(* Logix 5000 project; controller Sucrose_Main Emulate 5570 rev 20.12; software revision 20.01; part 2 of 30 *)

ADD_ON_INSTRUCTION QSI_Discrete_Device   (* revision 2.0 *)
// Revision note:
// Combined Discrete and Motor Starters into Single AOI
// Combined Feedback and No Feedback into Single AOI
// Added Config Param to select Feedback/No Feedback
// Added Config Param to Disable Output During Alarm
// Added Config Param to select "Energize"/"Start" Text
// Added Manual On Reset Logic During Alarm
// Added Zone & Device Specific Alarm Ack Logic
// Added Zone Manual Mode Enable Logic
// Help:
// Discrete Outputs Devices such as:
// Motors and Pumps on Starters, Solenoid Valves (Non FV and Non Analog Controlled), Beacons, Horns, Solenoids, etc.
VAR_OUTPUT
   DO_Energize : BOOL; {required}   // Alias to OutputCard to Energize DO
END_VAR
VAR_INPUT
   DI_Energized_Feedback : BOOL; {required}   // Alias to Input Card to Confirm Device is Energized
   DI_Disconnect_OK_Feedback : BOOL; {required}   // Alias to Input Card to Confirm Disconnect is OK
   ALM_ACK : BOOL; {required}   // Alias to Zone Master Alarm Acknowledge
   MM_Enable : BOOL; {required}   // Alias to Zone Master Manual Mode Enable
   Config_Energized_Feedback : BOOL := 1; {visible}   // Config Whether Device has Energized Feedback (0= No, 1= Yes) Note: Alarm Disabled if No Feedback
   Config_Disconnect_Feedback : BOOL := 1; {visible}   // Config Whether Device has Disconnect Feedback (0 = No, 1 = Yes)
   Config_Energized_Text : BOOL := 1; {visible}   // Configure Device HMI Popup Text (0="Started" {Motors, Pumps}; 1="Energized" {Most Devices}
   Config_MO_ResetOnAlarm : BOOL := 1; {visible}   // Configure Whether .MO Bit Turns Off when Device Alarm Condition Exists
   Config_OutputDisable_OnAlarm : BOOL; {visible}   // Configure Whether Device OutputTurns Off when Device Alarm Condition Exists
   Config_TMR_Alm_Preset_ms : DINT; {visible}   // Configure Device AlarmTimer Preset In Milliseconds
   Config_TMR_Off_Preset_ms : DINT; {visible}   // Configure Delay Stop Timer Preset In Milliseconds
   Config_TMR_On_Preset_ms : DINT; {visible}   // Configure Delay Start Timer Preset In Milliseconds
   HMI_MM : BOOL; {visible}   // Manual Mode Bit From HMI
   HMI_MO : BOOL; {visible}   // Manual On Bit From HMI
   HMI_ALM_ACK : BOOL;   // AOI Device Specific Alarm Acknowledge From HMI
END_VAR
VAR_OUTPUT
   HMI_Alarmed : BOOL;   // Alarm Status To HMI
   HMI_Energized : BOOL;   // Energized Status To HMI
   HMI_Disconnect_OK : BOOL;   // Disconnect Off Status To HMI
END_VAR
VAR_INPUT
   Energize_Permissive : BOOL;   // Energize Permissive Interlock From Logic
   Energize_Enable : BOOL;   // Energize Enable Interlock From Logic
END_VAR
VAR_OUTPUT
   ALM : BOOL; {visible}   // Device Alarm
END_VAR
VAR_INPUT
   Comment : BOOL;   // Comment for Description Rung to Start Each Routine
   Unused_Input_BOOL : BOOL;   // Trash Tag For Required AOI Input Variables That Are Unused for Current Device (Type Boolean)
END_VAR
VAR_OUTPUT
   Unused_Output_BOOL : BOOL;   // Trash Tag For Required AOI Output Variables That Are Unused for Current Device (Type Boolean)
END_VAR
VAR
   ONS : BOOL[32];
   TMR_Alm : TIMER; {access None}
   TMR_On : TIMER; {access None}
   TMR_Off : TIMER; {access None}
END_VAR

ROUTINE Logic   (* ladder *)
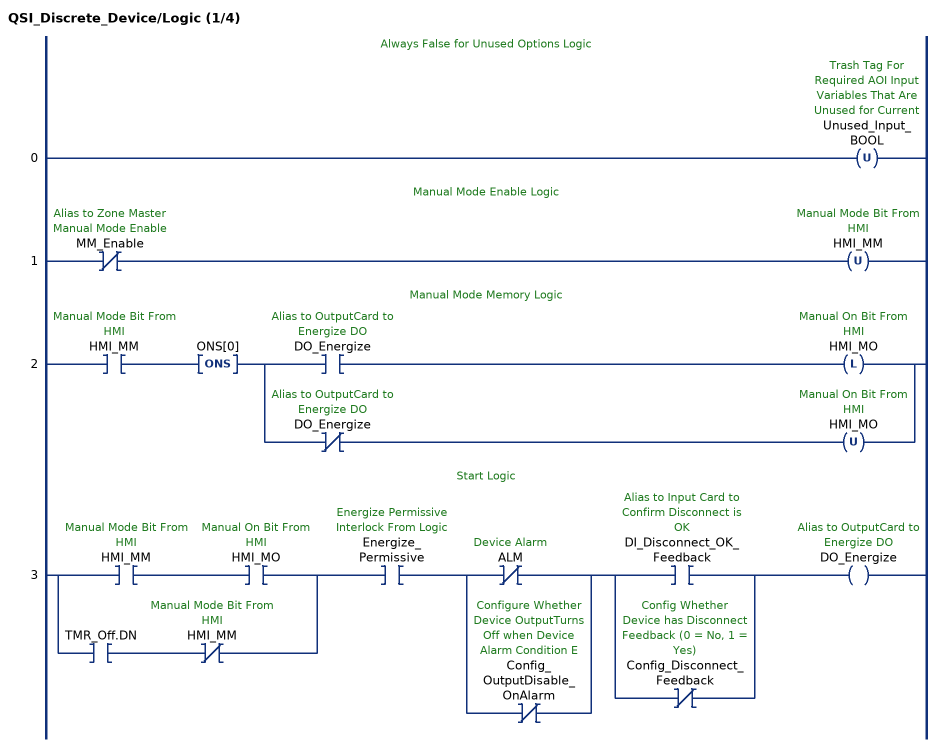
   // Always False for Unused Options Logic
   0: OTU(Unused_Input_BOOL);
   // Manual Mode Enable Logic
   1: XIO(MM_Enable)OTU(HMI_MM);
   // Manual Mode Memory Logic
   2: XIC(HMI_MM)ONS(ONS[0])[XIC(DO_Energize) OTL(HMI_MO) ,XIO(DO_Energize) OTU(HMI_MO) ];
   // Start Logic
   3: [XIC(HMI_MM) XIC(HMI_MO) ,XIC(TMR_Off.DN) XIO(HMI_MM) ]XIC(Energize_Permissive)[XIO(ALM) ,XIO(Config_OutputDisable_OnAlarm) ][XIC(DI_Disconnect_OK_Feedback) ,XIO(Config_Disconnect_Feedback) ]OTE(DO_Energize);
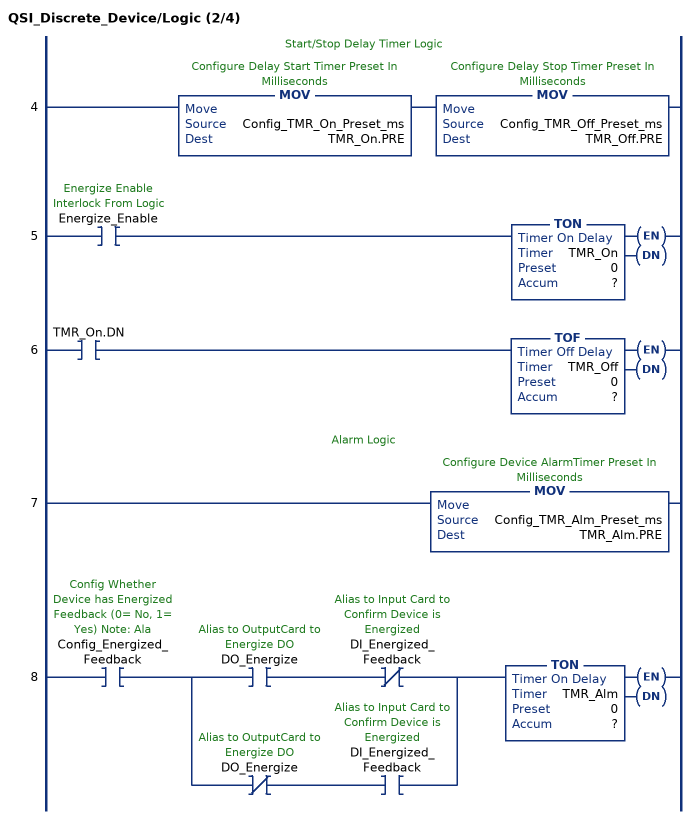
   // Start/Stop Delay Timer Logic
   4: MOV(Config_TMR_On_Preset_ms,TMR_On.PRE)MOV(Config_TMR_Off_Preset_ms,TMR_Off.PRE);
   5: XIC(Energize_Enable)TON(TMR_On,?,?);
   6: XIC(TMR_On.DN)TOF(TMR_Off,?,?);
   // Alarm Logic
   7: MOV(Config_TMR_Alm_Preset_ms,TMR_Alm.PRE);
   8: XIC(Config_Energized_Feedback)[XIC(DO_Energize) XIO(DI_Energized_Feedback) ,XIO(DO_Energize) XIC(DI_Energized_Feedback) ]TON(TMR_Alm,?,?);
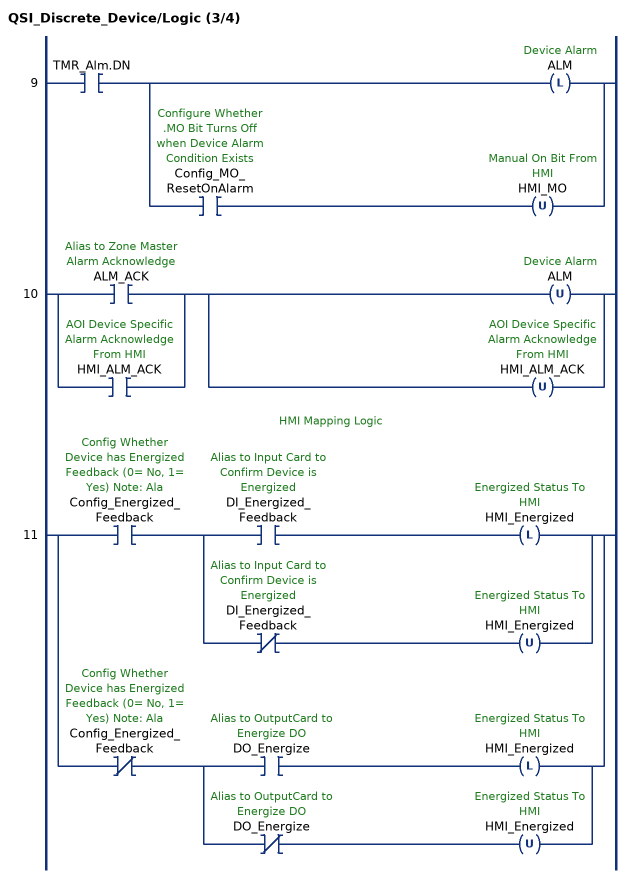
   9: XIC(TMR_Alm.DN)[OTL(ALM) ,XIC(Config_MO_ResetOnAlarm) OTU(HMI_MO) ];
   10: [XIC(ALM_ACK) ,XIC(HMI_ALM_ACK) ][OTU(ALM) ,OTU(HMI_ALM_ACK) ];
   // HMI Mapping Logic
   11: [XIC(Config_Energized_Feedback) [XIC(DI_Energized_Feedback) OTL(HMI_Energized) ,XIO(DI_Energized_Feedback) OTU(HMI_Energized) ] ,XIO(Config_Energized_Feedback) [XIC(DO_Energize) OTL(HMI_Energized) ,XIO(DO_Energize) OTU(HMI_Energized) ] ];
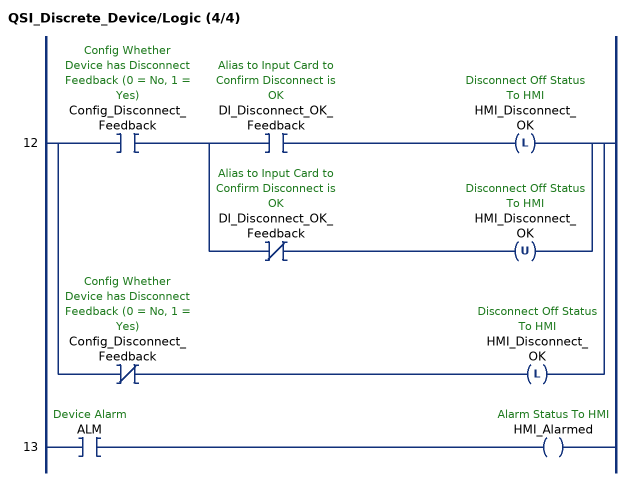
   12: [XIC(Config_Disconnect_Feedback) [XIC(DI_Disconnect_OK_Feedback) OTL(HMI_Disconnect_OK) ,XIO(DI_Disconnect_OK_Feedback) OTU(HMI_Disconnect_OK) ] ,XIO(Config_Disconnect_Feedback) OTL(HMI_Disconnect_OK) ];
   13: XIC(ALM)OTE(HMI_Alarmed);
END_ROUTINE
END_ADD_ON_INSTRUCTION

ADD_ON_INSTRUCTION QSI_Flow_Valve   (* revision 2.0 *)
// Revision note:
// Combined al Non-Analog Flow Valves  into Single AOI
// Combined Feedback and No Feedback into Single AOI
// Added Config Param to select N.O. or N.C. Valve
// Added Config Param to select Opened & Closed Feedback or No Feedback
// Added Manual On Reset Logic During Alarm
// Added Zone & Device Specific Alarm Ack Logic
// Added Zone Manual Mode Enable Logic
// Help:
// Discrete Flow Valves with and without feedback, and with and without Seat Lifts such as:
// Mix Proof, Stop Valves, and other Flow Valves
VAR_OUTPUT
   DO_Energize : BOOL; {required}   // Alias to OutputCard to Energize DO
   DO_USL_Energize : BOOL; {required}   // Alias to OutputCard to Energize Upper Seat Lift DO
   DO_LSL_Energize : BOOL; {required}   // Alias to OutputCard to Energize Lower Seat Lift DO
END_VAR
VAR_INPUT
   DI_Opened_Feedback : BOOL; {required}   // Alias to Input Card to Confirm Device is at Opened Position
   DI_Closed_Feedback : BOOL; {required}   // Alias to Input Card to Confirm Device is at Closed Position
   ALM_ACK : BOOL; {required}   // Alias to Zone Master Alarm Acknowledge
   MM_Enable : BOOL; {required}   // Alias to Zone Master Manual Mode Enable
   Config_NO_Valve : BOOL; {visible}   // Configure Whether Valve is Normally Closed (0 = N.C., 1 = N.O.)
   Config_Opened_Feedback : BOOL := 1; {visible}   // Config Whether Device has Opened Feedback (0= No, 1= Yes) Note: Alarm Disabled if No Feedback
   Config_Closed_Feedback : BOOL := 1; {visible}   // Config Whether Device has Closed Feedback (0= No, 1= Yes) Note: Alarm Disabled if No Feedback
   Config_MO_ResetOnAlarm : BOOL := 1; {visible}   // Configure Whether .MO Bit Turns Off when Device Alarm Condition Exists
   Config_TMR_Alm_Preset_ms : DINT; {visible}   // Configure Device AlarmTimer Preset In Milliseconds
   Config_TMR_Off_Preset_ms : DINT; {visible}   // Configure Delay Stop Timer Preset In Milliseconds
   Config_TMR_On_Preset_ms : DINT; {visible}   // Configure Delay Start Timer Preset In Milliseconds
   HMI_MM : BOOL; {visible}   // Manual Mode Bit From HMI
   HMI_MO : BOOL; {visible}   // Manual On Bit From HMI
   HMI_USL_MO : BOOL; {visible}   // Upper Seat Lift Manual On Bit From HMI
   HMI_LSL_MO : BOOL; {visible}   // Lower Seat Lift Manual On Bit From HMI
   HMI_ALM_ACK : BOOL;   // AOI Device Specific Alarm Acknowledge From HMI
END_VAR
VAR_OUTPUT
   HMI_Alarmed : BOOL;   // Alarm Status To HMI
   HMI_Opened : BOOL;   // Opened Status To HMI
   HMI_Closed : BOOL;   // Closed Status To HMI
END_VAR
VAR_INPUT
   Energize_Permissive : BOOL;   // Energize Permissive Interlock From Logic
   USL_Permissive : BOOL;   // Upper Seat Lift Permissive Interlock From Logic
   LSL_Permissive : BOOL;   // Lower Seat Lift Permissive Interlock From Logic
   Energize_Enable : BOOL;   // Energize Enable Interlock From Logic
   USL_Enable : BOOL;   // Upper Seat Lift Enable Interlock From Logic
   LSL_Enable : BOOL;   // Lower Seat Lift Enable Interlock From Logic
END_VAR
VAR_OUTPUT
   ALM : BOOL; {visible}   // Device Alarm
END_VAR
VAR_INPUT
   Comment : BOOL;   // Comment for Description Rung to Start Each Routine
   Unused_Input_BOOL : BOOL;   // Trash Tag For Required AOI Input Variables That Are Unused for Current Device (Type Boolean)
END_VAR
VAR_OUTPUT
   Unused_Output_BOOL : BOOL;   // Trash Tag For Required AOI Output Variables That Are Unused for Current Device (Type Boolean)
END_VAR
VAR
   ONS : BOOL[32];
   TMR_Alm : TIMER; {access None}
   TMR_On : TIMER; {access None}
   TMR_Off : TIMER; {access None}
END_VAR

ROUTINE Logic   (* ladder *)
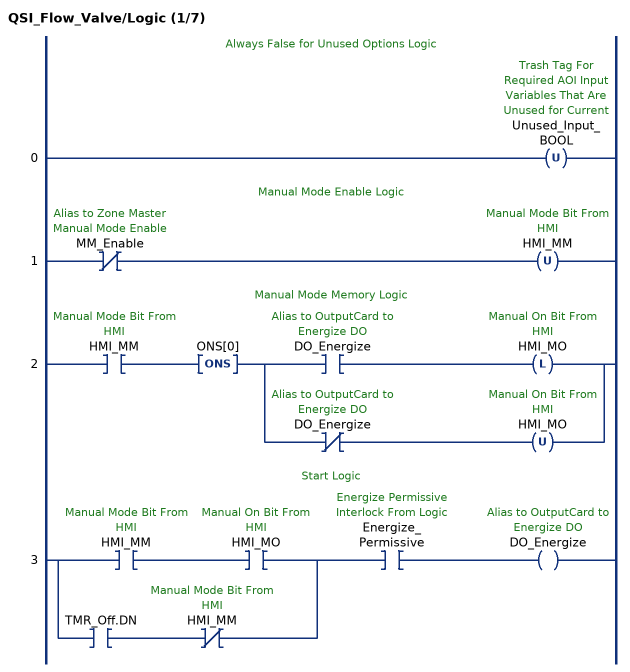
   // Always False for Unused Options Logic
   0: OTU(Unused_Input_BOOL);
   // Manual Mode Enable Logic
   1: XIO(MM_Enable)OTU(HMI_MM);
   // Manual Mode Memory Logic
   2: XIC(HMI_MM)ONS(ONS[0])[XIC(DO_Energize) OTL(HMI_MO) ,XIO(DO_Energize) OTU(HMI_MO) ];
   // Start Logic
   3: [XIC(HMI_MM) XIC(HMI_MO) ,XIC(TMR_Off.DN) XIO(HMI_MM) ]XIC(Energize_Permissive)OTE(DO_Energize);
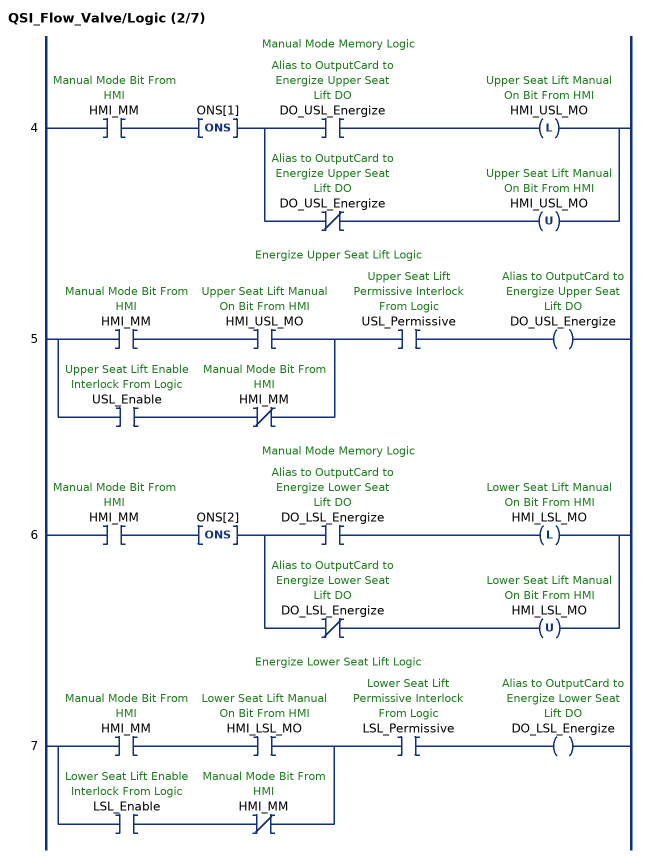
   // Manual Mode Memory Logic
   4: XIC(HMI_MM)ONS(ONS[1])[XIC(DO_USL_Energize) OTL(HMI_USL_MO) ,XIO(DO_USL_Energize) OTU(HMI_USL_MO) ];
   // Energize Upper Seat Lift Logic
   5: [XIC(HMI_MM) XIC(HMI_USL_MO) ,XIC(USL_Enable) XIO(HMI_MM) ]XIC(USL_Permissive)OTE(DO_USL_Energize);
   // Manual Mode Memory Logic
   6: XIC(HMI_MM)ONS(ONS[2])[XIC(DO_LSL_Energize) OTL(HMI_LSL_MO) ,XIO(DO_LSL_Energize) OTU(HMI_LSL_MO) ];
   // Energize Lower Seat Lift Logic
   7: [XIC(HMI_MM) XIC(HMI_LSL_MO) ,XIC(LSL_Enable) XIO(HMI_MM) ]XIC(LSL_Permissive)OTE(DO_LSL_Energize);
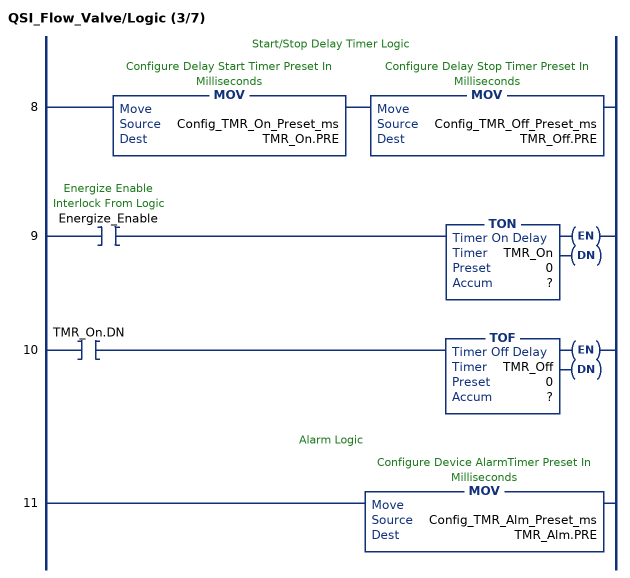
   // Start/Stop Delay Timer Logic
   8: MOV(Config_TMR_On_Preset_ms,TMR_On.PRE)MOV(Config_TMR_Off_Preset_ms,TMR_Off.PRE);
   9: XIC(Energize_Enable)TON(TMR_On,?,?);
   10: XIC(TMR_On.DN)TOF(TMR_Off,?,?);
   // Alarm Logic
   11: MOV(Config_TMR_Alm_Preset_ms,TMR_Alm.PRE);
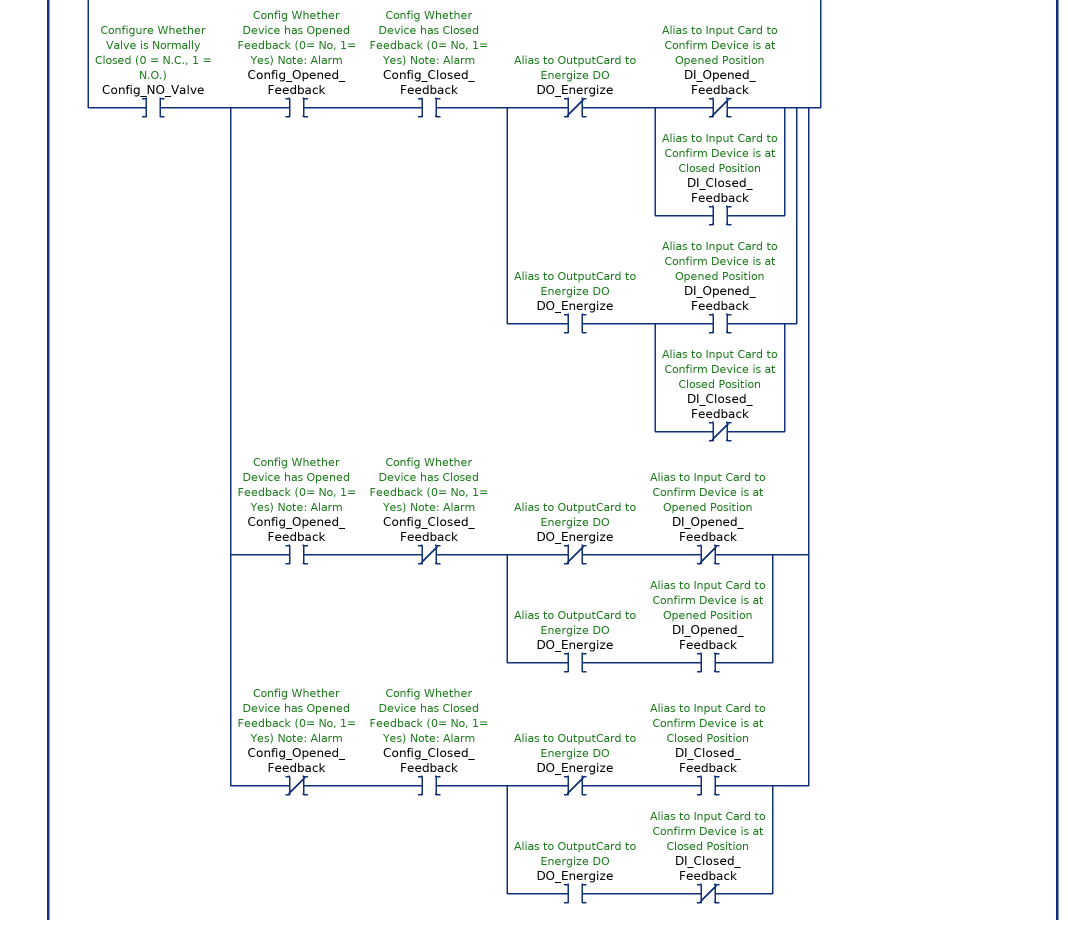
   12: XIO(DO_USL_Energize)XIO(DO_LSL_Energize)[XIO(Config_NO_Valve) [XIC(Config_Opened_Feedback) XIC(Config_Closed_Feedback) [XIC(DO_Energize) [XIO(DI_Opened_Feedback) ,XIC(DI_Closed_Feedback) ] ,XIO(DO_Energize) [XIC(DI_Opened_Feedback) ,XIO(DI_Closed_Feedback) ] ] ,XIC(Config_Opened_Feedback) XIO(Config_Closed_Feedback) [XIC(DO_Energize) XIO(DI_Opened_Feedback) ,XIO(DO_Energize) XIC(DI_Opened_Feedback) ] ,XIO(Config_Opened_Feedback) XIC(Config_Closed_Feedback) [XIC(DO_Energize) XIC(DI_Closed_Feedback) ,XIO(DO_Energize) XIO(DI_Closed_Feedback) ] ] ,XIC(Config_NO_Valve) [XIC(Config_Opened_Feedback) XIC(Config_Closed_Feedback) [XIO(DO_Energize) [XIO(DI_Opened_Feedback) ,XIC(DI_Closed_Feedback) ] ,XIC(DO_Energize) [XIC(DI_Opened_Feedback) ,XIO(DI_Closed_Feedback) ] ] ,XIC(Config_Opened_Feedback) XIO(Config_Closed_Feedback) [XIO(DO_Energize) XIO(DI_Opened_Feedback) ,XIC(DO_Energize) XIC(DI_Opened_Feedback) ] ,XIO(Config_Opened_Feedback) XIC(Config_Closed_Feedback) [XIO(DO_Energize) XIC(DI_Closed_Feedback) ,XIC(DO_Energize) XIO(DI_Closed_Feedback) ] ] ]TON(TMR_Alm,?,?);
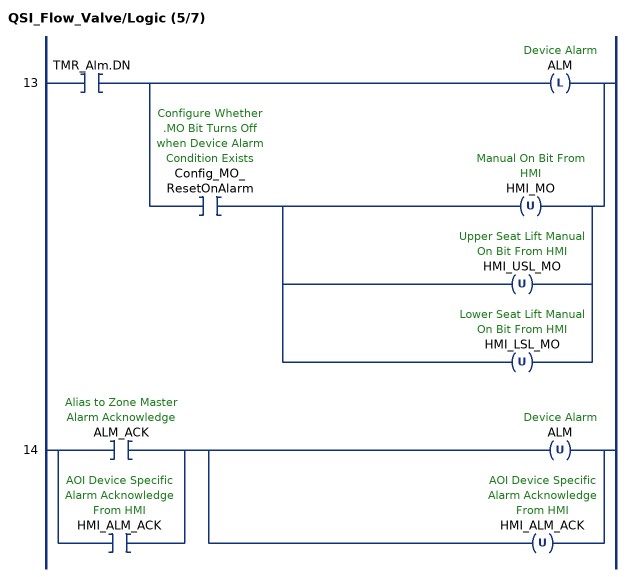
   13: XIC(TMR_Alm.DN)[OTL(ALM) ,XIC(Config_MO_ResetOnAlarm) [OTU(HMI_MO) ,OTU(HMI_USL_MO) ,OTU(HMI_LSL_MO) ] ];
   14: [XIC(ALM_ACK) ,XIC(HMI_ALM_ACK) ][OTU(ALM) ,OTU(HMI_ALM_ACK) ];
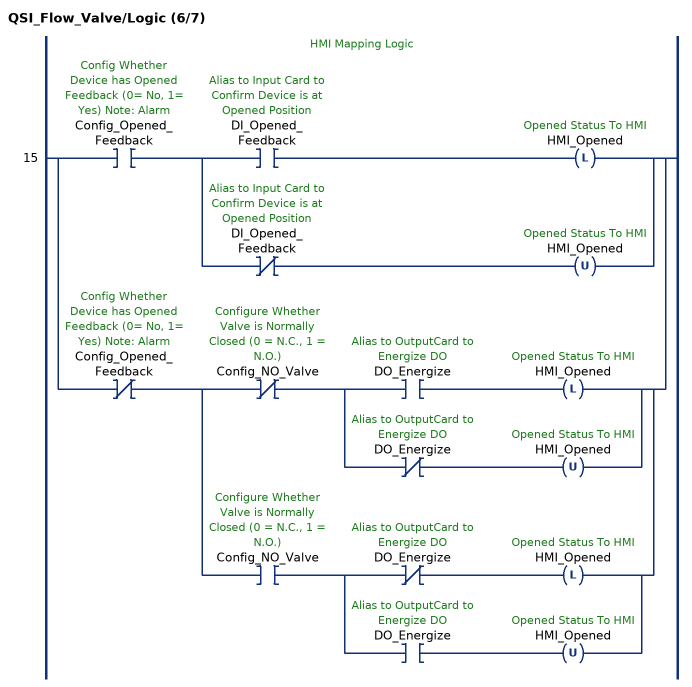
   // HMI Mapping Logic
   15: [XIC(Config_Opened_Feedback) [XIC(DI_Opened_Feedback) OTL(HMI_Opened) ,XIO(DI_Opened_Feedback) OTU(HMI_Opened) ] ,XIO(Config_Opened_Feedback) [XIO(Config_NO_Valve) [XIC(DO_Energize) OTL(HMI_Opened) ,XIO(DO_Energize) OTU(HMI_Opened) ] ,XIC(Config_NO_Valve) [XIO(DO_Energize) OTL(HMI_Opened) ,XIC(DO_Energize) OTU(HMI_Opened) ] ] ];
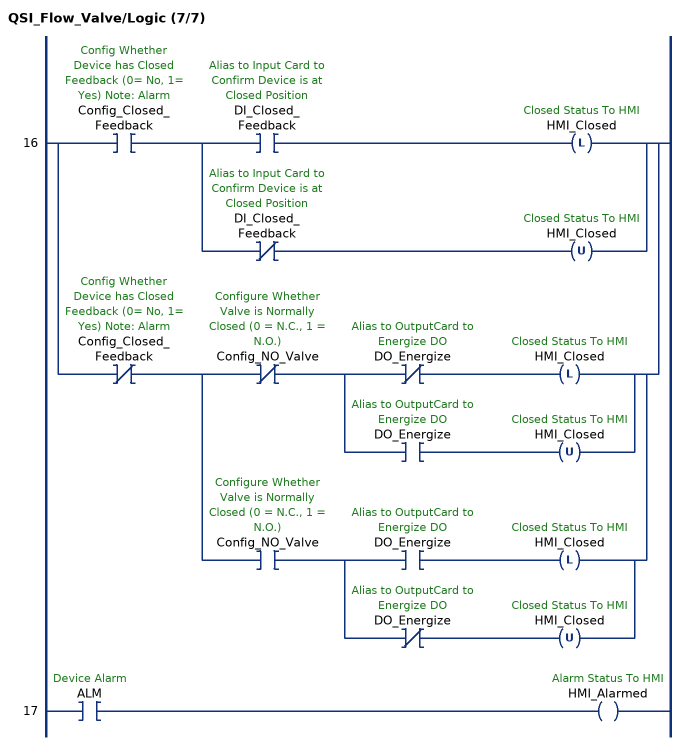
   16: [XIC(Config_Closed_Feedback) [XIC(DI_Closed_Feedback) OTL(HMI_Closed) ,XIO(DI_Closed_Feedback) OTU(HMI_Closed) ] ,XIO(Config_Closed_Feedback) [XIO(Config_NO_Valve) [XIO(DO_Energize) OTL(HMI_Closed) ,XIC(DO_Energize) OTU(HMI_Closed) ] ,XIC(Config_NO_Valve) [XIC(DO_Energize) OTL(HMI_Closed) ,XIO(DO_Energize) OTU(HMI_Closed) ] ] ];
   17: XIC(ALM)OTE(HMI_Alarmed);
END_ROUTINE
END_ADD_ON_INSTRUCTION

VAR_GLOBAL   (* controller tags *)
   AI_E21_0 : REAL[8];   // Analog Input EN2T_FLX 192.168.1.21
        [0]   // FIT-93-04-01 AIR INTEGRITY SUPPLY FLOW METER
        [1]   // PIT-23-05-01 PRE FILTER TRAIN 1 INLET PRESSURE TRANSMITTER
        [2]   // PIT-23-05-02 PRE FILTER TRAIN 1 OUTLET PRESSURE TRANSMITTER
        [3]   // PIT-23-05-03 FINAL FILTER TRAIN 1 INLET PRESSURE TRANSMITTER
        [4]   // PIT-23-05-04 FINAL FILTER TRAIN 1 OUTLET PRESSURE TRANSMITTER
        [5]   // PIT-23-06-01 PRE FILTER TRAIN 2 INLET PRESSURE TRANSMITTER
        [6]   // PIT-23-06-02 PRE FILTER TRAIN 2 OUTLET PRESSURE TRANSMITTER
        [7]   // PIT-23-06-03 FINAL FILTER TRAIN 2 INLET PRESSURE TRANSMITTER
   AI_E21_1 : REAL[8];   // Analog Input EN2T_FLX 192.168.1.21
        [0]   // PIT-23-06-04 FINAL FILTER TRAIN 2 OUTLET PRESSURE TRANSMITTER
        [1]   // PIT-93-04-01 AIR INTEGRITY TEST SUPPLY PRESSURE TRANSMITTER
        [2]   // TIT-74-05-01 PRE FILTRATION TRAIN 1 VENT TEMPERATURE TRANSMITTER
        [3]   // TIT-74-05-02 PRE FILTRATION TRAIN 1 STEAM TEMPERATURE TRANSMITTER
        [4]   // TIT-74-05-03 FINAL FILTRATION TRAIN 1 VENT TEMPERATURE TRANSMITTER
        [5]   // TIT-74-05-04 FINAL FILTRATION TRAIN 1 STEAM TEMPERATURE TRANSMITTER
        [6]   // TIT-74-06-01 PRE FILTRATION TRAIN 2 VENT TEMPERATURE TRANSMITTER
        [7]   // TIT-74-06-02 PRE FILTRATION TRAIN 2 STEAM TEMPERATURE TRANSMITTER
   AI_E21_2 : REAL[8];   // Analog Input EN2T_FLX 192.168.1.21
        [0]   // TIT-74-06-03 FINAL FILTRATION TRAIN 2 VENT TEMPERATURE TRANSMITTER
        [1]   // TIT-74-06-04 FINAL FILTRATION TRAIN 2 STEAM TEMPERATURE TRANSMITTER
        [2]   // AT-15-05-01 BRIX METER
        [3]   // SPARE SPARE ANALOG INPUT
        [4]   // SPARE SPARE ANALOG INPUT
        [5]   // SPARE SPARE ANALOG INPUT
        [6]   // SPARE SPARE ANALOG INPUT
        [7]   // SPARE SPARE ANALOG INPUT
   AI_E23_0 : REAL[8];   // Analog Input EN2T_FLX 192.168.1.23
        [0]   // LT-23-01-01 SUCROSE TANK #1 LEVEL TRANSMITTER
        [1]   // PIT-93-01-01 STERILE AIR TANK #1 AIR BLANKET PRESSURE TRANSMITTER
        [2]   // TIT-93-01-01 STERILE AIR TANK #1 AIR BLANKET TEMPERATURE TRANSMITTER
        [3]   // TIT-23-01-01 SUCROSE TANK #1 TEMPERATURE TRANSMITTER
        [4]   // LT-23-02-01 SUCROSE TANK #2 LEVEL TRANSMITTER
        [5]   // PIT-93-02-01 STERILE AIR TANK #2 AIR BLANKET PRESSURE TRANSMITTER
        [6]   // TIT-93-02-01 STERILE AIR TANK #2 AIR BLANKET TEMPERATURE TRANSMITTER
        [7]   // TIT-23-02-01 SUCROSE TANK #2 TEMPERATURE TRANSMITTER
   AI_E23_1 : REAL[8] := ([1] := 1320.1686, [2] := 58.190662, [3] := 0.10700389);   // Analog Input EN2T_FLX 192.168.1.23
        [0]   // TIT-74-03-01 SUCROSE TANK #1 STEAM SIP TANK BLANKETING TEMPERATURE TRANSMITTER
        [1]   // AT-91-01-01 AIR DRYER OUTLET DEW POINT TRANSMITTER
        [2]   // TIT-92-03-01 TANK AIR BLANKETING HEATER TEMPERATURE TRANSMITTER
        [3]   // FIT-23-01-01 SUCROSE HEADER FLOW RATE
        [4]   // LT-23-03-01 SUCROSE TANK #3 LEVEL TRANSMITTER
        [5]   // PIT-93-03-01 STERILE AIR TANK #3 AIR BLANKET PRESSURE TRANSMITTER
        [6]   // TIT-93-03-01 STERILE AIR TANK #3 AIR BLANKET TEMPERATURE TRANSMITTER
        [7]   // TIT-23-03-01 SUCROSE TANK #3 TEMPERATURE TRANSMITTER
   AI_E23_2 : REAL[8];   // Analog Input EN2T_FLX 192.168.1.23
        [0]   // TIT-74-03-02 SUCROSE TANK #2 STEAM SIP BLANKET TEMP TRANSMITTER
        [1]   // TIT-74-03-03 SUCROSE TANK #3 STEAM SIP BLANKET TEMP TRANSMITTER
        [2]   // SPARE ANALOG INPUT
        [3]   // SPARE ANALOG INPUT
        [4]   // SPARE ANALOG INPUT
        [5]   // SPARE ANALOG INPUT
        [6]   // SPARE ANALOG INPUT
        [7]   // SPARE ANALOG INPUT
   AI_E25_0 : REAL[8] := ([0] := 0.10700389, [1] := 0.3015564);   // Analog Input EN2T_FLX 192.168.1.25
        [0]   // FIT-23-00-10 MASS FLOW METER FOR RECEIVING PUMP P-23-00-10
        [1]   // FIT-23-00-20 MASS FLOW METER FOR RECEIVING PUMP P-23-00-20
        [2]   // TIT-XX-XX-XX SUCROSE RECEIVING BUILDING TEMPERATURE
        [3]   // SPARE SPARE ANALOG INPUT
        [4]   // SPARE SPARE ANALOG INPUT
        [5]   // SPARE SPARE ANALOG INPUT
        [6]   // SPARE SPARE ANALOG INPUT
        [7]   // SPARE SPARE ANALOG INPUT
   Alarm_ACK_Master_Timer : TIMER := (PRE := 2000);
   Alarm_ACK_Sucrose : BOOL;
   CIPRemote : Area_Program := (TMR_Logic[6].PRE := 10000, TMR_Logic[7].PRE := 10000, TMR_Logic[8].PRE := 10000, TMR_Logic[9].PRE := 10000, TMR_Logic[14].PRE := 10000, TMR_Logic[15].PRE := 10000, TMR_Logic[16].PRE := 10000, TMR_Logic[18].PRE := 10000, TMR_Logic[19].PRE := 10000, TMR_Logic[20].PRE := 10000);
        .BIT_HMI[0].0   // TANK 1 CIP YELLOW STATUS
        .BIT_LOGIC[0].0   // PIG VALVE PULSING BIT
        .BIT_HMI[0].1   // TANK 1 CIP RED STATUS
        .BIT_HMI[0].2   // TANK 2 CIP YELLOW STATUS
        .BIT_HMI[0].3   // TANK 2 CIP RED STATUS
        .BIT_HMI[0].4   // TANK 3 CIP YELLOW STATUS
        .BIT_HMI[0].5   // TANK 3 CIP RED STATUS
   ClearFault_Master : BOOL;
   ClearFault_Master_TMR : TIMER;
   CR13582_AOI : QSI_Discrete_Device := (MM_Enable := 1, Config_Energized_Text := 1, Config_MO_ResetOnAlarm := 1, Config_TMR_Alm_Preset_ms := 10000, Energize_Permissive := 1, Comment := 1);   // CR-13582 SUCROSE RECEIVING PUMP #1 SEAL WATER VALVE
   CR13584_AOI : QSI_Discrete_Device := (MM_Enable := 1, Config_Energized_Text := 1, Config_MO_ResetOnAlarm := 1, Config_TMR_Alm_Preset_ms := 10000, HMI_Disconnect_OK := 1, Energize_Permissive := 1, Comment := 1);   // CR-13584 SUCROSE RECEIVING PUMP #2 SEAL WATER VALVE
   DATE_TIME : Date_Time;
   DI_E20_0 : ALIAS FOR FLX_E20:0:I;   // Discrete Input EN2T_FLX 192.168.1.20
        .0   // ZSO-23-04-11 SUCROSE TANK #1 TO TRANSFER PUMP #1 MIX PROOF VALVE OPEN
        .1   // ZSC-23-04-11 SUCROSE TANK #1 TO TRANSFER PUMP #1 MIX PROOF VALVE CLOSED
        .2   // ZSO-23-04-12 SUCROSE TANK #2 TO TRANSFER PUMP #1 MIX PROOF VALVE OPEN
        .3   // ZSC-23-04-12 SUCROSE TANK #2 TO TRANSFER PUMP #1 MIX PROOF VALVE CLOSED
        .4   // ZSO-23-04-13 SUCROSE TANK #3 TO TRANSFER PUMP #1 MIX PROOF VALVE OPEN
        .5   // ZSC-23-04-13 SUCROSE TANK #3 TO TRANSFER PUMP #1 MIX PROOF VALVE CLOSED
        .6   // ZSO-23-04-41 SUCROSE TRANSFER PUMP #1 DISCHARGE TO FILTRATION OPEN
        .7   // ZSC-23-04-41 SUCROSE TRANSFER PUMP #1 DISCHARGE TO FILTRATION CLOSED
        .8   // ZSO-23-04-42 SUCROSE TRANSFER PUMP #2 DISCHARGE TO FILTRATION OPEN
        .9   // ZSC-23-04-42 SUCROSE TRANSFER PUMP #2 DISCHARGE TO FILTRATION CLOSED
        .10   // ZSO-61-05-01 CIP SUPPLY TO FILTRATION AND RING MAIN MIX PROOF VALVE OPEN
        .11   // ZSC-61-05-01 CIP SUPPLY TO FILTRATION AND RING MAIN MIX PROOF VALVE CLOSED
        .12   // ZSO-23-04-21 SUCROSE TANK #1 TO TRANSFER PUMP #2 MIX PROOF VALVE OPEN
        .13   // ZSC-23-04-21 SUCROSE TANK #1 TO TRANSFER PUMP #2 MIX PROOF VALVE CLOSED
        .14   // ZSO-23-04-22 SUCROSE TANK #2 TO TRANSFER PUMP #2 MIX PROOF VALVE OPEN
        .15   // ZSC-23-04-22 SUCROSE TANK #2 TO TRANSFER PUMP #2 MIX PROOF VALVE CLOSED
   DI_E20_1 : ALIAS FOR FLX_E20:1:I;   // Discrete Input EN2T_FLX 192.168.1.20
        .0   // ZSO-23-04-23 SUCROSE TANK #3 TO TRANSFER PUMP #2 MIX PROOF VALVE OPEN
        .1   // ZSC-23-04-23 SUCROSE TANK #3 TO TRANSFER PUMP #2 MIX PROOF VALVE CLOSED
        .2   // ZSO-62-01-01 SUCROSE TANK #1 TO CIP RETURN MIX PROOF VALVE OPEN
        .3   // ZSC-62-01-01 SUCROSE TANK #1 TO CIP RETURN MIX PROOF VALVE CLOSED
        .4   // ZSO-62-02-01 SUCROSE TANK #2 TO CIP RETURN MIX PROOF VALVE OPEN
        .5   // ZSC-62-02-01 SUCROSE TANK #2 TO CIP RETURN MIX PROOF VALVE CLOSED
        .6   // ZSO-62-03-01 SUCROSE TANK #3 TO CIP RETURN PUMP MIX PROOF VALVE OPEN
        .7   // ZSC-62-03-01 SUCROSE TANK #3 TO CIP RETURN PUMP MIX PROOF VALVE CLOSED
        .8   // ZSO-62-04-01 TRANSFER PUMP #1 TO CIP RETURN MIX PROOF VALVE OPEN
        .9   // ZSC-62-04-01 TRANSFER PUMP #1 TO CIP RETURN MIX PROOF VALVE CLOSED
        .10   // ZSO-62-04-02 TRANSFER PUMP #2 TO CIP RETURN MIX PROOF VALVE OPEN
        .11   // ZSC-62-04-02 TRANSFER PUMP #2 TO CIP RETURN MIX PROOF VALVE CLOSED
        .12   // SPARE 24VDC INPUT
        .13   // SPARE 24VDC INPUT
        .14   // SPARE 24VDC INPUT
        .15   // SPARE 24VDC INPUT
   DI_E20_2 : ALIAS FOR FLX_E20:2:I;   // Discrete Input EN2T_FLX 192.168.1.20
        .0   // 1400-ADS-12019 SUCROSE TRANSFER PUMP #1, P-23-04-01, DISCONNECT OK
        .1   // 1400-ADS-12027 SUCROSE TRANSFER PUMP #2, P-23-04-02, DISCONNECT OK
        .2   // 1400-ADS-12035 CIP RETURN PUMP, P-62-01-01, DISCONNECT OK
        .3   // SPARE 24VDC INPUT
        .4   // SPARE 24VDC INPUT
        .5   // SPARE 24VDC INPUT
        .6   // SPARE 24VDC INPUT
        .7   // SPARE 24VDC INPUT
        .8   // SPARE 24VDC INPUT
        .9   // SPARE 24VDC INPUT
        .10   // SPARE 24VDC INPUT
        .11   // SPARE 24VDC INPUT
        .12   // SPARE 24VDC INPUT
        .13   // SPARE 24VDC INPUT
        .14   // SPARE 24VDC INPUT
        .15   // CR-16016 E-STOP MCR-1
   DI_E22_0 : ALIAS FOR FLX_E22:0:I;   // Discrete Input EN2T_FLX 192.168.1.22
        .0   // ZSO-23-05-01-OPEN PRE FILTER TRAIN 1 INLET VALVE OPEN
        .1   // ZSC-23-05-01-CLOSED PRE FILTER TRAIN 1 INLET VALVE CLOSED
        .2   // ZSO-23-05-06-OPEN PRE FILTER TRAIN 1 OUTLET VALVE OPEN
        .3   // ZSC-23-05-06-CLOSED PRE FILTER TRAIN 1 OUTLET VALVE CLOSED
        .4   // ZSO-23-05-08-OPEN FINAL FILTER TRAIN 1 INLET VALVE OPEN
        .5   // ZSC-23-05-08-CLOSED FINAL FILTER TRAIN 1 INLET VALVE CLOSED
        .6   // ZSO-23-05-13-OPEN FINAL FILTER TRAIN 1 OUTLET VALVE OPEN
        .7   // ZSC-23-05-13-CLOSED FINAL FILTER TRAIN 1 OUTLET VALVE CLOSED
        .8   // ZSO-23-06-01-OPEN PRE FILTER TRAIN 2 INLET VALVE OPEN
        .9   // ZSC-23-06-01-CLOSED PRE FILTER TRAIN 2 INLET VALVE CLOSED
        .10   // ZSO-23-06-06-OPEN PRE FILTER TRAIN 2 OUTLET VALVE OPEN
        .11   // ZSC-23-06-06-CLOSED PRE FILTER TRAIN 2 OUTLET VALVE CLOSED
        .12   // ZSO-23-06-08-OPEN FINAL FILTER TRAIN 2 INLET VALVE OPEN
        .13   // ZSC-23-06-08-CLOSED FINAL FILTER TRAIN 2 INLET VALVE CLOSED
        .14   // ZSO-23-06-13-OPEN FINAL FILTER TRAIN 2 OUTLET VALVE OPEN
        .15   // ZSC-23-06-13-CLOSED FINAL FILTER TRAIN 2 OUTLET VALVE CLOSED
   DI_E22_1 : ALIAS FOR FLX_E22:1:I;   // Discrete Input EN2T_FLX 192.168.1.22
        .0   // SPARE SPARE 24VDC INPUT
        .1   // SPARE SPARE 24VDC INPUT
        .2   // SPARE SPARE 24VDC INPUT
        .3   // SPARE SPARE 24VDC INPUT
        .4   // SPARE SPARE 24VDC INPUT
        .5   // SPARE SPARE 24VDC INPUT
        .6   // SPARE SPARE 24VDC INPUT
        .7   // SPARE SPARE 24VDC INPUT
        .8   // SPARE SPARE 24VDC INPUT
        .9   // SPARE SPARE 24VDC INPUT
        .10   // SPARE SPARE 24VDC INPUT
        .11   // SPARE SPARE 24VDC INPUT
        .12   // SPARE SPARE 24VDC INPUT
        .13   // SPARE SPARE 24VDC INPUT
        .14   // SPARE SPARE 24VDC INPUT
        .15   // SPARE SPARE 24VDC INPUT
   DI_E23_3 : ALIAS FOR FLX_E23:3:I;   // Discrete Input EN2T_FLX 192.168.1.23
        .0   // LSH-93-01-01 SUCROSE TANK #1 LEVEL SWITCH HIGH
        .1   // ZSC-93-11-01 STERILE AIR SUCROSE TANK #1 RUPTURE DISK SENSOR
        .2   // ZSC-61-01-01 SUCROSE TANK #1 MANWAY CIP JUMPER POXIMITY SWITCH
        .3   // HTR-76-01-01 UTILITY HOT WATER TANK #1 ELECTRIC HEATER CONTROLLER STATUS
        .4   // LSH-93-02-01 SUCROSE TANK #2 LEVEL SWITCH HIGH
        .5   // ZSC-93-12-01 STERILE AIR SUCROSE TANK #2 RUPTURE DISK SENSOR
        .6   // ZSC-61-02-01 SUCROSE TANK #2 MANWAY CIP JUMPER POXIMITY SWITCH
        .7   // HTR-76-02-01 UTILITY HOT WATER TANK #2 ELECTRIC HEATER CONTROLLER STATUS
        .8   // LSH-93-03-01 SUCROSE TANK #3 LEVEL SWITCH HIGH
        .9   // ZSC-93-13-01 STERILE AIR SUCROSE TANK #3 RUPTURE DISK SENSOR
        .10   // ZSC-61-03-01 SUCROSE TANK #3 MANWAY CIP JUMPER POXIMITY SWITCH
        .11   // HTR-76-03-01 UTILITY HOT WATER TANK #3 ELECTRIC HEATER CONTROLLER STATUS
        .12   // FLT-91-03-01 AIR DRYER ALARM
        .13   // SPARE 24VDC INPUT
        .14   // SPARE 24VDC INPUT
        .15   // SPARE 24VDC INPUT
   DI_E23_4 : ALIAS FOR FLX_E23:4:I;   // Discrete Input EN2T_FLX 192.168.1.23
        .0   // ZSO-23-00-06 RETURN PIG TO LAUNCHER VALVE V7 OPEN
        .1   // ZSC-23-00-06 RETURN PIG TO LAUNCHER VALVE V7 CLOSED
        .2   // ZSO-23-00-07 RETURN PIG TO LAUNCHER VALVE V6 OPEN
        .3   // ZSC-23-00-07 RETURN PIG TO LAUNCHER VALVE V6 CLOSED
        .4   // ZSC-23-00-13 PIG AT RECEIVING STATION PROX SWITCH
        .5   // SPARE 24VDC INPUT
        .6   // ZSO-23-01-01 SUCROSE RECEIVING TO SUCROSE TANK #1 VALVE OPEN
        .7   // ZSC-23-01-01 SUCROSE RECEIVING TO SUCROSE TANK #1 VALVE CLOSED
        .8   // ZSO-23-01-04 SUCROSE RETURN TO SUCROSE TANK #1 VALVE OPEN
        .9   // ZSC-23-01-04 SUCROSE RETURN TO SUCROSE TANK #1 VALVE CLOSED
        .10   // ZSO-23-02-01 SUCROSE RECEIVING TO SUCROSE TANK #2 VALVE OPEN
        .11   // ZSC-23-02-01 SUCROSE RECEIVING TO SUCROSE TANK #2 VALVE CLOSED
        .12   // ZSO-23-02-04 SUCROSE RETURN TO SUCROSE TANK #2 VALVE OPEN
        .13   // ZSC-23-02-04 SUCROSE RETURN TO SUCROSE TANK #2 VALVE CLOSED
        .14   // ZSO-23-03-01 SUCROSE RECEIVING TO SUCROSE TANK #3 VALVE OPEN
        .15   // ZSC-23-03-01 SUCROSE RECEIVING TO SUCROSE TANK #3 VALVE CLOSED
   DI_E23_5 : ALIAS FOR FLX_E23:5:I;   // Discrete Input EN2T_FLX 192.168.1.23
        .0   // ZSO-23-03-04 SUCROSE RETURN TO SUCROSE TANK #3 VALVE OPEN
        .1   // ZSC-23-03-04 SUCROSE RETURN TO SUCROSE TANK #3 VALVE CLOSED
        .2   // ZSO-61-01-01 CIP SUPPLY TO SUCROSE TANK #1 VALVE OPEN
        .3   // ZSC-61-01-01 CIP SUPPLY TO SUCROSE TANK #1 VALVE CLOSED
        .4   // ZSO-61-02-01 CIP SUPPLY TO SUCROSE TANK #2 VALVE OPEN
        .5   // ZSC-61-02-01 CIP SUPPLY TO SUCROSE TANK #2 VALVE CLOSED
        .6   // ZSO-61-03-01 CIP SUPPLY TO SUCROSE TANK #3 VALVE OPEN
        .7   // ZSC-61-03-01 CIP SUPPLY TO SUCROSE TANK #3 VALVE CLOSED
        .8   // ZSO-61-04-01 VALVE MANIFOLD TO SUCROSE TRANSFER PUMP #1 VALVE OPEN
        .9   // ZSC-61-04-01 VALVE MANIFOLD TO SUCROSE TRANSFER PUMP #1 VALVE CLOSED
        .10   // ZSO-61-04-02 VALVE MANIFOLD TO SUCROSE TRANSFER PUMP #2 VALVE OPEN
        .11   // ZSC-61-04-02 VALVE MANIFOLD TO SUCROSE TRANSFER PUMP #2 VALVE CLOSED
        .12   // ZSO-62-00-01 SUCROSE RECEIVING TO CIP RETURN VALVE OPEN
        .13   // ZSC-62-00-01 SUCROSE RECEIVING TO CIP RETURN VALVE CLOSED
        .14   // ZSO-62-07-01 SUCROSE RING MAIN RETURN TO CIP RETURN VALVE VALVE OPEN
        .15   // ZSC-62-07-01 SUCROSE RING MAIN RETURN TO CIP RETURN VALVE VALVE CLOSED
   DI_E23_6 : ALIAS FOR FLX_E23:6:I;   // Discrete Input EN2T_FLX 192.168.1.23
        .0   // SPARE 24VDC INPUT
        .1   // SPARE 24VDC INPUT
        .2   // SPARE 24VDC INPUT
        .3   // SPARE 24VDC INPUT
        .4   // SPARE 24VDC INPUT
        .5   // SPARE 24VDC INPUT
        .6   // SPARE 24VDC INPUT
        .7   // SPARE 24VDC INPUT
        .8   // SPARE 24VDC INPUT
        .9   // SPARE 24VDC INPUT
        .10   // SPARE 24VDC INPUT
        .11   // SPARE 24VDC INPUT
        .12   // SPARE 24VDC INPUT
        .13   // SPARE 24VDC INPUT
        .14   // SPARE 24VDC INPUT
        .15   // SPARE 24VDC INPUT
   DI_E25_2 : ALIAS FOR FLX_E25:2:I;   // Discrete Input EN2T_FLX 192.168.1.25
        .0   // ZSO-23-00-01 LAUNCH PIG VALVE V1 OPEN
        .1   // ZSC-23-00-01 LAUNCH PIG VALVE V1 CLOSED
        .2   // ZSO-23-00-02 LAUNCH PIG VALVE V2 OPEN
        .3   // ZSC-23-00-02 LAUNCH PIG VALVE V3 CLOSED
        .4   // ZSC-23-00-03.1 PIG MOVED FORWARD INTO LAUNCHING POSITION PROX SWITCH
        .5   // ZSC-23-00-03.2 PIG MOVED BACKWORDS INTO CIP POSITION PROX SWITCH
        .6   // ZSO-23-00-04 PIG RETENTION CYLINDER V4.1 OPEN
        .7   // ZSC-23-00-04 PIG RETENTION CYLINDER V4.1 CLOSED
        .8   // ZSO-23-00-05 PIG RETENTION CYLINDER V4.2 OPEN
        .9   // ZSC-23-00-05 PIG RETENTION CYLINDER V4.2 CLOSED
        .10   // ZSC-23-00-11 PIG IN CLEANING-PRODUCTION POSITION PROX SWITCH
        .11   // ZSC-23-00-12 PIG IN LAUNCHING POSITION PROX SWITCH
        .12   // SPARE SPARE 24VDC INPUT
        .13   // SPARE SPARE 24VDC INPUT
        .14   // SPARE SPARE 24VDC INPUT
        .15   // SPARE SPARE 24VDC INPUT
   DI_E25_3 : ALIAS FOR FLX_E25:3:I;   // Discrete Input EN2T_FLX 192.168.1.25
        .0   // ZSO-23-00-10 RECEIVING PUMP #1 TO SUCROSE VALVE MANIFOLD MIX PROOF VALVE OPEN
        .1   // ZSC-23-00-10 RECEIVING PUMP #1 TO SUCROSE VALVE MANIFOLD MIX PROOF VALVE CLOSED
        .2   // ZSO-23-00-20 RECEIVING PUMP #2 TO SUCROSE VALVE MANIFOLD MIX PROOF VALVE OPEN
        .3   // ZSC-23-00-20 RECEIVING PUMP #2 TO SUCROSE VALVE MANIFOLD MIX PROOF VALVE CLOSED
        .4   // ZSO-62-00-10 RECEIVING PUMP #1 TO CIP RETURN MIX PROOF VALVE OPEN
        .5   // ZSC-62-00-10 RECEIVING PUMP #1 TO CIP RETURN MIX PROOF VALVE CLOSED
        .6   // ZSO-62-00-20 RECEIVING PUMP #2 TO CIP RETURN MIX PROOF VALVE OPEN
        .7   // ZSC-62-00-20 RECEIVING PUMP #2 TO CIP RETURN MIX PROOF VALVE CLOSED
        .8   // ADS-12019 SUCROSE RECEIVING PUMP #1 P-23-00-10 DISCONNECT
        .9   // ADS-12027 SUCROSE RECEIVING PUMP #2 P-23-00-20 DISCONNECT
        .10   // SPARE SPARE 24VDC INPUT
        .11   // SPARE SPARE 24VDC INPUT
        .12   // SPARE SPARE 24VDC INPUT
        .13   // SPARE SPARE 24VDC INPUT
        .14   // SPARE SPARE 24VDC INPUT
        .15   // CR-16016 E-STOP MCR1
   DISCHARGE_NO_ALARM : BOOL;   // SUCROSE HEADER NO ACTIVE ALARMS FOR P_23_01_01 PATH
   DISCHARGE_NO_ALARM2 : BOOL;   // SUCROSE HEADER NO ACTIVE ALARMS FOR P_23_01_02 PATH
   DO_E20_3 : ALIAS FOR FLX_E20:3:O;   // Discrete Output EN2T_FLX 192.168.1.20
        .0   // FV-23-04-11-O SUCROSE TANK #1 TO TRANSFER PUMP #1 MIX PROOF VALVE OPEN
        .1   // FV-23-04-11-UL SUCROSE TANK #1 TO TRANSFER PUMP #1 MIX PROOF VALVE UPPER LIFT
        .2   // FV-23-04-11-LL SUCROSE TANK #1 TO TRANSFER PUMP #2 MIX PROOF VALVE LOWER LIFT
        .3   // FV-23-04-12-O SUCROSE TANK #2 TO TRANSFER PUMP #1 MIX PROOF VALVE OPEN
        .4   // FV-23-04-12-UL SUCROSE TANK #2 TO TRANSFER PUMP #1 MIX PROOF VALVE UPPER LIFT
        .5   // FV-23-04-12-LL SUCROSE TANK #2 TO TRANSFER PUMP #1 MIX PROOF VALVE LOWER LIFT
        .6   // FV-23-04-13-O SUCROSE TANK #3 TO TRANSFER PUMP #1 MIX PROOF VALVE OPEN
        .7   // FV-23-04-13-UL SUCROSE TANK #3 TO TRANSFER PUMP #1 MIX PROOF VALVE UPPER LIFT
        .8   // FV-23-04-13-LL SUCROSE TANK #3 TO TRANSFER PUMP #1 MIX PROOF VALVE LOWER LIFT
        .9   // FV-23-04-41-O SUCROSE TRANSFER PUMP #1 DISCHARGE TO FILTRATRION MIX PROOF VALVE OPEN
        .10   // FV-23-04-41-UL SUCROSE TRANSFER PUMP #1 DISCHARGE TO FILTRATRION MIX PROOF VALVE UPPER LIFT
        .11   // FV-23-04-41-LL SUCROSE TRANSFER PUMP #1 DISCHARGE TO FILTRATRION MIX PROOF VALVE LOWER LIFT
        .12   // FV-23-04-42-O SUCROSE TRANSFER PUMP #2 DISCHARGE TO FILTRATRION MIX PROOF VALVE OPEN
        .13   // FV-23-04-42-UL SUCROSE TRANSFER PUMP #2 DISCHARGE TO FILTRATRION MIX PROOF VALVE UPPER LIFT
        .14   // FV-23-04-42-LL SUCROSE TRANSFER PUMP #2 DISCHARGE TO FILTRATRION MIX PROOF VALVE LOWER LIFT
        .15   // SPARE 24VDC OUTPUT
   DO_E20_4 : ALIAS FOR FLX_E20:4:O;   // Discrete Output EN2T_FLX 192.168.1.20
        .0   // FV-61-05-01-O CIP SUPPLY TO FILTRATION AND RING MAIN MIX PROOF VALVE OPEN
        .1   // FV-61-05-01-UL CIP SUPPLY TO FILTRATION AND RING MAIN MIX PROOF VALVE UPER LIFT
        .2   // FV-61-05-01-LL CIP SUPPLY TO FILTRATION AND RING MAIN MIX PROOF VALVE LOWER LIFT
        .3   // FV-23-04-21-O SUCROSE TANK #1 TO TRANSFER PUMP #2 MIX PROOF VALVE OPEN
        .4   // FV-23-04-21-UL SUCROSE TANK #1 TO TRANSFER PUMP #2 MIX PROOF VALVE UPPER LIFT
        .5   // FV-23-04-21-LL SUCROSE TANK #1 TO TRANSFER PUMP #2 MIX PROOF VALVE LOWER LIFT
        .6   // FV-23-02-22-O SUCROSE TANK #2 TO TRANSFER PUMP #2 MIX PROOF VALVE OPEN
        .7   // FV-23-02-22-UL SUCROSE TANK #2 TO TRANSFER PUMP #2 MIX PROOF VALVE UPPER LIFT
        .8   // FV-23-02-22-LL SUCROSE TANK #2 TO TRANSFER PUMP #2 MIX PROOF VALVE LOWER LIFT
        .9   // FV-23-04-23-O SUCROSE TANK #3 TO TRANSFER PUMP #2 MIX PROOF VALVE OPEN
        .10   // FV-23-04-23-UL SUCROSE TANK #3 TO TRANSFER PUMP #2 MIX PROOF VALVE UPPER LIFT
        .11   // FV-23-04-23-LL SUCROSE TANK #3 TO TRANSFER PUMP #2 MIX PROOF VALVE LOWER LIFT
        .12   // FV-62-01-01-O SUCROSE TANK #1 TO CIP RETURN PUMP MIX PROOF VALVE OPEN
        .13   // FV-62-01-01-UL SUCROSE TANK #1 TO CIP RETURN PUMP MIX PROOF VALVE UPPER LIFT
        .14   // FV-62-01-01-LL SUCROSE TANK #1 TO CIP RETURN PUMP MIX PROOF VALVE LOWER LIFT
        .15   // SPARE 24VDC OUTPUT
   DO_E20_5 : ALIAS FOR FLX_E20:5:O;   // Discrete Output EN2T_FLX 192.168.1.20
        .0   // FV-62-02-01-O SUCROSE TANK #2 TO CIP RETURN PUMP MIX PROOF VALVE OPEN
        .1   // FV-62-02-01-UL SUCROSE TANK #2 TO CIP RETURN PUMP MIX PROOF VALVE UPPER LIFT
        .2   // FV-62-02-01-LL SUCROSE TANK #2 TO CIP RETURN PUMP MIX PROOF VALVE LOWER LIFT
        .3   // FV-62-03-01-O SUCROSE TANK #3 TO CIP RETURN PUMP MIX PROOF VALVE OPEN
        .4   // FV-62-03-01-UL SUCROSE TANK #3 TO CIP RETURN PUMP MIX PROOF VALVE UPPER LIFT
        .5   // FV-62-03-01-LL SUCROSE TANK #3 TO CIP RETURN PUMP MIX PROOF VALVE LOWER LIFT
        .6   // FV-62-04-01-O CIP RETURN PUMP #1 TO FILTER SYSTEM MIX PROOF VALVE OPEN
        .7   // FV-62-04-01-UL CIP RETURN PUMP #1 TO FILTER SYSTEM MIX PROOF VALVE UPPER LIFT
        .8   // FV-62-04-01-LL CIP RETURN PUMP #1 TO FILTER SYSTEM MIX PROOF VALVE LOWER LIFT
        .9   // FV-62-04-02-O CIP RETURN PUMP #2 TO FILTER SYSTEM MIX PROOF VALVE OPEN
        .10   // FV-62-04-02-UL CIP RETURN PUMP #2 TO FILTER SYSTEM MIX PROOF VALVE UPPER LIFT
        .11   // FV-62-04-02-LL CIP RETURN PUMP #2 TO FILTER SYSTEM MIX PROOF VALVE LOWER LIFT
        .14   // SPARE 24VDC OUTPUT
        .15   // PBL-16040-01 RESET PB LIGHT
   DO_E20_6 : ALIAS FOR FLX_E20:6:O;   // Discrete Output EN2T_FLX 192.168.1.20
        .0   // FV-23-04-31 SUCROSE LOW POINT DRAIN VALVE @ TRANSFER PUMP #1
        .1   // FV-23-04-32 SUCROSE LOW POINT DRAIN VALVE @ TRANSFER PUMP #2
        .2   // FV-61-04-11 CIP SUPPLY TO TRANSFER PUMP #1 OR TO DRAIN DIVERT VALVE
        .3   // FV-61-04-12 CIP SUPPLY TO TRANSFER PUMP #2 OR TO DRAIN DIVERT VALVE
        .4   // FV-23-04-01 SUCROSE TANK #3 LOW POINT DRAIN
        .5   // FV-23-04-02 SUCROSE TANK #2 LOW POINT DRAIN
        .6   // FV-23-04-03 SUCROSE TANK #1 LOW POINT DRAIN
        .7   // FV-62-04-00 CIP RETURN LOW POINT DRAIN VALVE
        .8   // PSV-23-04-01 TRANSFER PUMP #1 BYPASS VALVE
        .9   // PSV-23-04-02 TRANSFER PUMP #2 BYPASS VALVE
        .10   // SPARE SV
        .11   // SPARE SV
        .12   // SPARE SV
        .13   // SPARE 24VDC OUTPUT
        .14   // SPARE 24VDC OUTPUT
        .15   // SPARE 24VDC OUTPUT
   DO_E20_7 : ALIAS FOR FLX_E20:7:O;   // Discrete Output EN2T_FLX 192.168.1.20
        .0   // SV-13-04-01 SUCROSE TRANSFER PUMP #1 SEAL WATER FLUSH VALVE
        .1   // SV-13-04-02 SUCROSE TRANSFER PUMP #2 SEAL WATER FLUSH VALVE
        .2   // SPARE RELAY OUTPUT
        .3   // SPARE RELAY OUTPUT
        .4   // SPARE RELAY OUTPUT
        .5   // SPARE RELAY OUTPUT
        .6   // SPARE RELAY OUTPUT
        .7   // SPARE RELAY OUTPUT
   DO_E22_2 : ALIAS FOR FLX_E22:2:O;   // Discrete Output EN2T_FLX 192.168.1.22
        .0   // FV-23-05-01-O PRE FILTER TRAIN 1 INLET VALVE OPEN
        .1   // FV-23-05-01-UL PRE FILTER TRAIN 1 INLET VALVE UPPER LIFT
        .2   // FV-23-05-01-LL PRE FILTER TRAIN 1 INLET VALVE LOWER LIFT
        .3   // FV-23-05-06-O PRE FILTER TRAIN 1 OUTLET VALVE OPEN
        .4   // FV-23-05-06-UL PRE FILTER TRAIN 1 OUTLET VALVE UPPER LIFT
        .5   // FV-23-05-06-LL PRE FILTER TRAIN 1 OUTLET VALVE LOWER LIFT
        .6   // FV-23-05-08-O FINAL FILTER TRAIN 1 INLET VALVE OPEN
        .7   // FV-23-05-08-UL FINAL FILTER TRAIN 1 INLET VALVE UPPER LIFT
        .8   // FV-23-05-08-LL FINAL FILTER TRAIN 1 INLET VALVE LOWER LIFT
        .9   // FV-23-05-13-O FINAL FILTER TRAIN 1 OUTLET VALVE OPEN
        .10   // FV-23-05-13-UL FINAL FILTER TRAIN 1 OUTLET VALVE UPPER LIFT
        .11   // FV-23-05-13-LL FINAL FILTER TRAIN 1 OUTLET VALVE LOWER LIFT
        .12   // FV-23-06-01-O PRE FILTER TRAIN 2 INLET VALVE OPEN
        .13   // FV-23-06-01-UL PRE FILTER TRAIN 2 INLET VALVE UPPER LIFT
        .14   // FV-23-06-01-LL PRE FILTER TRAIN 2 INLET VALVE LOWER LIFT
        .15   // SPARE SPARE 24VDC OUTPUT
   DO_E22_3 : ALIAS FOR FLX_E22:3:O;   // Discrete Output EN2T_FLX 192.168.1.22
        .0   // FV-23-06-06-O PRE FILTER TRAIN 2 OUTLET VALVE OPEN
        .1   // FV-23-06-06-UL PRE FILTER TRAIN 2 OUTLET VALVE UPPER LIFT
        .2   // FV-23-06-06-LL PRE FILTER TRAIN 2 OUTLET VALVE LOWER LIFT
        .3   // FV-23-06-08-O FINAL FILTER TRAIN 2 INLET VALVE OPEN
        .4   // FV-23-06-08-UL FINAL FILTER TRAIN 2 INLET VALVE UPPER LIFT
        .5   // FV-23-06-08-LL FINAL FILTER TRAIN 2 INLET VALVE LOWER LIFT
        .6   // FV-23-06-13-O FINAL FILTER TRAIN 2 OUTLET VALVE OPEN
        .7   // FV-23-06-13-UL FINAL FILTER TRAIN 2 OUTLET VALVE UPPER LIFT
        .8   // FV-23-06-13-LL FINAL FILTER TRAIN 2 OUTLET VALVE LOWER LIFT
        .9   // SPARE SPARE 24VDC OUTPUT
        .10   // SPARE SPARE 24VDC OUTPUT
        .11   // SPARE SPARE 24VDC OUTPUT
        .12   // SPARE SPARE 24VDC OUTPUT
        .13   // SPARE SPARE 24VDC OUTPUT
        .14   // SPARE SPARE 24VDC OUTPUT
        .15   // SPARE SPARE 24VDC OUTPUT
   DO_E22_4 : ALIAS FOR FLX_E22:4:O;   // Discrete Output EN2T_FLX 192.168.1.22
        .0   // FV-14-05-01 PRE FILTER TRAIN 1 SUPPLY VALVE
        .1   // FV-14-05-02 FINAL FILTER TRAIN 1 SUPPLY VALVE
        .2   // FV-14-05-03 HOT WATER LOW POINT DRAIN VALVE
        .3   // FV-14-06-01 PRE FILTER TRAIN 2 SUPPLY VALVE
        .4   // FV-14-06-02 FINAL FILTER TRAIN 2 SUPPLY VALVE
        .5   // FV-15-05-01 DIVERT TO SCRAP OR TO DRAIN VALVE
        .6   // FV-23-05-00 SUCROSE LOW POINT DRAIN VALVE
        .7   // FV-23-05-02 PRE FILTER TRAIN 1 INLET LOW POINT DRAIN VALVE
        .8   // FV-23-05-03 PRE FILTER TRAIN 1 INLET LOW POINT DRAIN VALVE
        .9   // FV-23-05-04 PRE FILTER TRAIN 1 OUTLET LOW POINT DRAIN VALVE
        .10   // FV-23-05-05 PRE FILTER TRAIN 1 OUTLET LOW POINT DRAIN VALVE
        .11   // FV-23-05-09 FINAL FILTER TRAIN 1 INLET LOW POINT DRAIN VALVE
        .12   // SPARE SV SPARE SV
        .13   // SPARE SV SPARE SV
        .14   // SPARE 24VDC OUTPUT
        .15   // SPARE 24VDC OUTPUT
   DO_E22_5 : ALIAS FOR FLX_E22:5:O;   // Discrete Output EN2T_FLX 192.168.1.22
        .0   // FV-23-05-10 FINAL FILTER TRAIN 1 INLET LOW POINT DRAIN VALVE
        .1   // FV-23-05-11 FINAL FILTER TRAIN 1 OUTLET LOW POINT DRAIN VALVE
        .2   // FV-23-05-12 FINAL FILTER TRAIN 1 OUTLET LOW POINT DRAIN VALVE
        .3   // FV-23-06-02 PRE FILTER TRAIN 2 INLET LOW POINT DRAIN VALVE
        .4   // FV-23-06-03 PRE FILTER TRAIN 2 INLET LOW POINT DRAIN VALVE
        .5   // FV-23-06-04 PRE FILTER TRAIN 2 OUTLET LOW POINT DRAIN VALVE
        .6   // FV-23-06-05 PRE FILTER TRAIN 2 OUTLET LOW POINT DRAIN VALVE
        .7   // FV-23-06-07 LOW POINT DRAIN VALVE
        .8   // FV-23-06-09 FINAL FILTER TRAIN 2 INLET LOW POINT DRAIN VALVE
        .9   // FV-23-06-10 FINAL FILTER TRAIN 2 INLET LOW POINT DRAIN VALVE
        .10   // FV-23-06-11 FINAL FILTER TRAIN 2 OUTLET LOW POINT DRAIN VALVE
        .11   // FV-23-06-12 FINAL FILTER TRAIN 2 OUTLET LOW POINT DRAIN VALVE
        .12   // SPARE SV SPARE SV
        .13   // SPARE SV SPARE SV
        .14   // SPARE 24VDC OUTPUT
        .15   // SPARE 24VDC OUTPUT
   DO_E22_6 : ALIAS FOR FLX_E22:6:O;   // Discrete Output EN2T_FLX 192.168.1.22
        .0   // FV-74-04-01 SIP SUPPLY VALVE
        .1   // FV-74-05-01 SIP SUPPLY TO PRE FILTER TRAIN 1 VALVE
        .2   // FV-74-05-02 SIP SUPPLY TO FINAL FILTER TRAIN 1 VALVE
        .3   // FV-74-06-01 SIP SUPPLY TO PRE FILTER TRAIN 2 VALVE
        .4   // FV-74-06-02 SIP SUPPLY TO FINAL FILTER TRAIN 2 VALVE
        .5   // FV-75-05-01 TRP-75-05-01 ISOLATION VALVE
        .6   // FV-75-05-02 TRP-75-05-02 ISOLATION VALVE
        .7   // FV-75-05-03 TRP-75-05-03 ISOLATION VALVE
        .8   // FV-75-05-04 TRP-75-05-04 ISOLATION VALVE
        .9   // FV-75-06-01 TRP-75-06-01 ISOLATION VALVE
        .10   // FV-75-06-02 TRP-75-06-02 ISOLATION VALVE
        .11   // FV-75-06-03 TRP-75-06-03 ISOLATION VALVE
        .12   // FV-93-05-11 PRE FILTER TRAIN 1 AIR BLOW OUTLET
        .13   // FV-93-05-12 FINAL FILTER TRAIN 1 AIR BLOW OUTLET
        .14   // SPARE SPARE 24VDC OUTPUT
        .15   // SPARE SPARE 24VDC OUTPUT
   DO_E22_7 : ALIAS FOR FLX_E22:7:O;   // Discrete Output EN2T_FLX 192.168.1.22
        .0   // FV-75-06-04 TRP-75-06-04 ISOLATION VALVE
        .1   // FV-92-05-01 FLT-23-05-01 VENT VALVE
        .2   // FV-92-05-02 FLT-23-05-02 VENT VALVE
        .3   // FV-92-06-01 FLT-23-06-01 VENT VALVE
        .4   // FV-93-04-01 FLT-93-04-01 INLET VALVE
        .5   // FV-93-05-01 PRE FILTER TRAIN 1 AIR BLOW INLET
        .6   // FV-93-05-03 INTEGRITY TEST TO SUPPLY TO FINAL FILTER TRAIN 1 VALVE
        .7   // FV-93-05-02 FINAL FILTER TRAIN 1 AIR BLOW VALVE
        .8   // FV-93-06-01 PRE FILTER TRAIN 2 AIR BLOW INLET
        .9   // FV-92-06-02 FLT-23-06-02 VENT VALVE
        .10   // FV-93-06-03 INTEGRITY TEST TO SUPPLY TO FINAL FILTER DRAIN VALVE
        .11   // FV-93-06-02 FINAL FILTER TRAIN 2 AIR BLOW OUTLET
        .12   // FV-93-06-11 PRE FILTER TRAIN 2 AIR BLOW OUTLET
        .13   // FV-93-06-12 FINAL FILTER TRAIN 2 AIR BLOW OUTLET
        .14   // SPARE SPARE 24VDC OUTPUT
        .15   // SPARE SPARE 24VDC OUTPUT
   DO_E24_0 : ALIAS FOR FLX_E24:0:O;   // Discrete Output EN2T_FLX 192.168.1.24
        .0   // FV-23-00-06 RETURN PIG TO LAUNCHER VALVE V7
        .1   // FV-23-00-07 RETURN PIG TO LAUNCHER VALVE V6
        .2   // FV-23-01-01-O SUCROSE RECEIVING TO SUCROSE TANK #1 VALVE OPEN
        .3   // FV-23-01-01-UL SUCROSE RECEIVING TO SUCROSE TANK #1 VALVE UPPER LIFT
        .4   // FV-23-01-01-LL SUCROSE RECEIVING TO SUCROSE TANK #1 VALVE LOWER LIFT
        .5   // FV-23-01-04-O SUCROSE RETURN TO SUCROSE TANK #1 VALVE OPEN
        .6   // FV-23-01-04-UL SUCROSE RETURN TO SUCROSE TANK #1 VALVE UPPER LIFT
        .7   // FV-23-01-04-LL SUCROSE RETURN TO SUCROSE TANK #1 VALVE LOWER LIFT
        .8   // FV-23-02-01-O SUCROSE RECEIVING TO SUCROSE TANK #2 VALVE OPEN
        .9   // FV-23-02-01-UL SUCROSE RECEIVING TO SUCROSE TANK #2 VALVE UPPER LIFT
        .10   // FV-23-02-01-LL SUCROSE RECEIVING TO SUCROSE TANK #2 VALVE LOWER LIFT
        .11   // FV-23-02-04-O SUCROSE RETURN TO SUCROSE TANK #2 VALVE OPEN
        .12   // FV-23-02-04-UL SUCROSE RETURN TO SUCROSE TANK #2 VALVE UPPER LIFT
        .13   // FV-23-02-04-LL SUCROSE RETURN TO SUCROSE TANK #2 VALVE LOWER LIFT
        .14   // SPARE 24VDC OUTPUT
        .15   // SPARE 24VDC OUTPUT
   DO_E24_1 : ALIAS FOR FLX_E24:1:O;   // Discrete Output EN2T_FLX 192.168.1.24
        .0   // FV-23-03-01-O SUCROSE RECEIVING TO SUCROSE TANK #3 VALVE OPEN
        .1   // FV-23-03-01-UL SUCROSE RECEIVING TO SUCROSE TANK #3 VALVE UPPER LIFT
        .2   // FV-23-03-01-LL SUCROSE RECEIVING TO SUCROSE TANK #3 VALVE LOWER LIFT
        .3   // FV-23-03-04-O SUCROSE RETURN TO SUCROSE TANK #3 VALVE OPEN
        .4   // FV-23-03-04-UL SUCROSE RETURN TO SUCROSE TANK #3 VALVE UPPER LIFT
        .5   // FV-23-03-04-LL SUCROSE RETURN TO SUCROSE TANK #3 VALVE LOWER LIFT
        .6   // FV-61-01-01-O CIP SUPPLY TO SUCROSE TANK #1 VALVE OPEN
        .7   // FV-61-01-01-UL CIP SUPPLY TO SUCROSE TANK #1 VALVE UPPER LIFT
        .8   // FV-61-01-01-LL CIP SUPPLY TO SUCROSE TANK #1 VALVE LOWER LIFT
        .9   // FV-61-02-01-O CIP SUPPLY TO SUCROSE TANK #2 VALVE OPEN
        .10   // FV-61-02-01-UL CIP SUPPLY TO SUCROSE TANK #2 VALVE UPPER LIFT
        .11   // FV-61-02-01-LL CIP SUPPLY TO SUCROSE TANK #2 VALVE LOWER LIFT
        .12   // FV-61-03-01-O CIP SUPPLY TO SUCROSE TANK #3 VALVE OPEN
        .13   // FV-61-03-01-UL CIP SUPPLY TO SUCROSE TANK #3 VALVE UPPER LIFT
        .14   // FV-61-03-01-LL CIP SUPPLY TO SUCROSE TANK #3 VALVE LOWER LIFT
        .15   // SPARE 24VDC OUTPUT
   DO_E24_2 : ALIAS FOR FLX_E24:2:O;   // Discrete Output EN2T_FLX 192.168.1.24
        .0   // FV-61-04-01-O VALVE MANIFOLD TO SUCROSE TRANSFER PUMP #1 VALVE OPEN
        .1   // FV-61-04-01-UL VALVE MANIFOLD TO SUCROSE TRANSFER PUMP #1 VALVE UPPER LIFT
        .2   // FV-61-04-01-LL VALVE MANIFOLD TO SUCROSE TRANSFER PUMP #1 VALVE LOWER LIFT
        .3   // FV-61-04-02-O VALVE MANIFOLD TO SUCROSE TRANSFER PUMP #2 VALVE OPEN
        .4   // FV-61-04-02-UL VALVE MANIFOLD TO SUCROSE TRANSFER PUMP #2 VALVE UPPER LIFT
        .5   // FV-61-04-02-LL VALVE MANIFOLD TO SUCROSE TRANSFER PUMP #2 VALVE LOWER LIFT
        .6   // FV-62-00-01-O SUCROSE RECEIVING TO CIP RETURN VALVE OPEN
        .7   // FV-62-00-01-UL SUCROSE RECEIVING TO CIP RETURN VALVE UPPER LIFT
        .8   // FV-62-00-01-LL SUCROSE RECEIVING TO CIP RETURN VALVE LOWER LIFT
        .9   // FV-62-07-01-O SUCROSE RING MAIN RETURN TO CIP RETURN VALVE VALVE OPEN
        .10   // FV-62-07-01-UL SUCROSE RING MAIN RETURN TO CIP RETURN VALVE VALVE UPPER LIFT
        .11   // FV-62-07-01-LL SUCROSE RING MAIN RETURN TO CIP RETURN VALVE VALVE LOWER LIFT
        .12   // HTR-92-03-01 COMPRESSED AIR TANK AIR BLANKETING HEATER
        .13   // SPARE 24VDC OUTPUT
        .14   // SPARE 24VDC OUTPUT
        .15   // SPARE 24VDC OUTPUT
   DO_E24_3 : ALIAS FOR FLX_E24:3:O;   // Discrete Output EN2T_FLX 192.168.1.24
        .0   // FV-23-01-02 SUCROSE TANK #1 INLET/SPRAYBALL VALVE
        .1   // FV-23-01-03 SUCROSE TANK #1 OUTLET VALVE
        .2   // FV-75-11-01 SUCROSE TANK #1 BLANKETING STEAM TRAP ISOLATION VALVE
        .3   // FV-93-11-01 STERILE AIR FLT-93-11-01 SHUT OFF VALVE
        .4   // FV-23-02-02 SUCROSE TANK #2 INLET/SPRAYBALL VALVE
        .5   // FV-23-02-03 SUCROSE TANK #2 OUTLET VALVE
        .6   // FV-75-12-01 SUCROSE TANK #2 BLANKETING STEAM TRAP ISOLATION VALVE
        .7   // FV-93-12-01 STERILE AIR FLT-93-12-01 SHUT OFF VALVE
        .8   // SPARE SV
        .9   // SPARE SV
        .10   // FV-23-03-02 SUCROSE TANK #3 INLET/SPRAYBALL VALVE
        .11   // FV-23-03-03 SUCROSE TANK #3 OUTLET VALVE
        .12   // FV-75-13-01 SUCROSE TANK #3 BLANKETING STEAM TRAP ISOLATION VALVE
        .13   // FV-93-13-01 STERILE AIR FLT-93-13-01 SHUT OFF VALVE
        .14   // FV-75-14-01 CONDENSATE TANK BLANKETING STEAM TRAP ISOLATION VALVE
        .15   // FV-92-03-01 INSTRUMENT AIR HEATER ISOLATION VALVE
   DO_E24_4 : ALIAS FOR FLX_E24:4:O;   // Discrete Output EN2T_FLX 192.168.1.24
        .0   // FV-74-03-01 STEAM SIP SUPPLY VALVE
        .1   // SPARE SV
        .2   // SPARE SV
        .3   // SPARE SV
        .4   // SPARE 24VDC OUTPUT
        .5   // SPARE 24VDC OUTPUT
        .6   // SPARE 24VDC OUTPUT
        .7   // SPARE 24VDC OUTPUT
        .8   // SPARE 24VDC OUTPUT
        .9   // SPARE 24VDC OUTPUT
        .10   // SPARE 24VDC OUTPUT
        .11   // SPARE 24VDC OUTPUT
        .12   // SPARE 24VDC OUTPUT
        .13   // SPARE 24VDC OUTPUT
        .14   // SPARE 24VDC OUTPUT
        .15   // SPARE 24VDC OUTPUT
   DO_E24_5 : ALIAS FOR FLX_E24:5:O;   // Discrete Output EN2T_FLX 192.168.1.24
        .0   // HTR-76-01-01 SUCROSE TANK #1 UTILITY HOT WATER ELECTRIC HEATER ENABLE
        .1   // HTR-76-02-01 SUCROSE TANK #2 UTILITY HOT WATER ELECTRIC HEATER ENABLE
        .2   // HTR-76-03-01 SUCROSE TANK #3 UTILITY HOT WATER ELECTRIC HEATER ENABLE
        .3   // SPARE RELAY OUTPUT
        .4   // SPARE RELAY OUTPUT
        .5   // SPARE RELAY OUTPUT
        .6   // SPARE RELAY OUTPUT
        .7   // SPARE RELAY OUTPUT
   DO_E24_6 : ALIAS FOR FLX_E24:6:O;   // Discrete Output EN2T_FLX 192.168.1.24
        .0   // SV-93-11-01 STERILE AIR AUTO VENT FOR FLT-93-11-01 SOLENOID VALVE
        .1   // SV-93-11-02 STERILE AIR AUTO DRAIN FOR FLT-93-11-01 SOLENOID VALVE
        .2   // SV-93-12-01 STERILE AIR AUTO VENT FOR FLT-93-12-01 SOLENOID VALVE
        .3   // SV-93-12-02 STERILE AIR AUTO DRAIN FOR FLT-93-12-01 SOLENOID VALVE
        .4   // SV-93-13-01 STERILE AIR AUTO VENT FOR FLT-93-13-01 SOLENOID VALVE
        .5   // SV-93-13-02 STERILE AIR AUTO DRAIN FOR FLT-93-13-01 SOLENOID VALVE
        .6   // SPARE RELAY OUTPUT
        .7   // SPARE RELAY OUTPUT
   DO_E25_4 : ALIAS FOR FLX_E25:4:O;   // Discrete Output EN2T_FLX 192.168.1.25
        .0   // FV-23-00-01 LAUNCH PIG VALVE V1
        .1   // FV-23-00-02 LAUNCH PIG VALVE V2
        .2   // FV-23-00-04 PIG RETENTION CYLINDER V4.1
        .3   // FV-23-00-03.1 MOVE PIG BACKWARDS INTO CIP/PRODUCTION POSITION
        .4   // FV-23-00-05 PIG RETENTION CYLINDER V4.2
        .5   // FV-23-00-03.2 MOVE PIG FORWARD INTO LAUNCHING POSITION
        .6   // SPARE SPARE 24VDC OUTPUT
        .7   // SPARE SPARE 24VDC OUTPUT
        .8   // SPARE SPARE 24VDC OUTPUT
        .9   // SPARE SPARE 24VDC OUTPUT
        .10   // PSV-23-00-10 SUCROSE RECEIVING PUMP #1 BYPASS VALVE
        .11   // PSV-23-00-20 SUCROSE RECEIVING PUMP #2 BYPASS VALVE
        .12   // FV-61-00-10 CIP SUPPLY TO RECEIVING PUMP #1
        .13   // FV-61-00-20 CIP SUPPLY TO RECEIVING PUMP #2
        .14   // FV-61-00-30 CIP LOW POINT DRAIN
        .15   // SPARE SV SPARE SV
   DO_E25_5 : ALIAS FOR FLX_E25:5:O;   // Discrete Output EN2T_FLX 192.168.1.25
        .0   // FV-23-00-10-O RECEIVING PUMP #1 TO SUCROSE VALVE MANIFOLD MIX PROOF VALVE OPEN
        .1   // FV-23-00-10-UL RECEIVING PUMP #1 TO SUCROSE VALVE MANIFOLD MIX PROOF VALVE UPPER LIFT
        .2   // FV-23-00-10-LL RECEIVING PUMP #1 TO SUCROSE VALVE MANIFOLD MIX PROOF VALVE LOWER LIFT
        .3   // FV-23-00-20-O RECEIVING PUMP #2 TO SUCROSE VALVE MANIFOLD MIX PROOF VALVE OPEN
        .4   // FV-23-00-20-UL RECEIVING PUMP #2 TO SUCROSE VALVE MANIFOLD MIX PROOF VALVE UPPER LIFT
        .5   // FV-23-00-20-LL RECEIVING PUMP #2 TO SUCROSE VALVE MANIFOLD MIX PROOF VALVE LOWER LIFT
        .6   // FV-62-00-10-O RECEIVING PUMP #1 TO CIP RETURN MIX PROOF VALVE OPEN
        .7   // FV-62-00-10-UL RECEIVING PUMP #1 TO CIP RETURN MIX PROOF VALVE UPPER LIFT
        .8   // FV-62-00-10-LL RECEIVING PUMP #1 TO CIP RETURN MIX PROOF VALVE LOWER LIFT
        .9   // FV-62-00-20-O RECEIVING PUMP #2 TO CIP RETURN MIX PROOF VALVE OPEN
        .10   // FV-62-00-20-UL RECEIVING PUMP #2 TO CIP RETURN MIX PROOF VALVE UPPER LIFT
        .11   // FV-62-00-20-LL RECEIVING PUMP #2 TO CIP RETURN MIX PROOF VALVE LOWER LIFT
        .12   // SPARE SPARE 24VDC OUTPUT
        .13   // PBL-16040-02 E-STOP CIRCUIT RESET LIGHT
        .14   // CR-13582 SUCROSE RECEIVING PUMP #1 SEAL WATER VALVE
        .15   // CR-13584 SUCROSE RECEIVING PUMP #2 SEAL WATER VALVE
   FV140501_AOI : QSI_Flow_Valve := (MM_Enable := 1, Config_MO_ResetOnAlarm := 1, Config_TMR_Alm_Preset_ms := 10000, HMI_Closed := 1, Energize_Permissive := 1, Comment := 1);   // FV-14-05-01 PRE FILTER TRAIN 1 SUPPLY VALVE
   FV140502_AOI : QSI_Flow_Valve := (MM_Enable := 1, Config_MO_ResetOnAlarm := 1, Config_TMR_Alm_Preset_ms := 10000, HMI_Closed := 1, Energize_Permissive := 1, Comment := 1);   // FV-14-05-02 FINAL FILTER TRAIN 1 SUPPLY VALVE
   FV140503_AOI : QSI_Flow_Valve := (MM_Enable := 1, Config_MO_ResetOnAlarm := 1, Config_TMR_Alm_Preset_ms := 10000, HMI_Closed := 1, Energize_Permissive := 1, Comment := 1);   // FV-14-05-03 HOT WATER LOW POINT DRAIN VALVE
   FV140601_AOI : QSI_Flow_Valve := (MM_Enable := 1, Config_MO_ResetOnAlarm := 1, Config_TMR_Alm_Preset_ms := 10000, HMI_Closed := 1, Energize_Permissive := 1, Comment := 1);   // FV-14-06-01 PRE FILTER TRAIN 2 SUPPLY VALVE
   FV140602_AOI : QSI_Flow_Valve := (MM_Enable := 1, Config_MO_ResetOnAlarm := 1, Config_TMR_Alm_Preset_ms := 10000, HMI_Closed := 1, Energize_Permissive := 1, Comment := 1);   // FV-14-06-02 FINAL FILTER TRAIN 2 SUPPLY VALVE
   FV150501_AOI : QSI_Flow_Valve := (MM_Enable := 1, Config_MO_ResetOnAlarm := 1, Config_TMR_Alm_Preset_ms := 10000, HMI_Closed := 1, Energize_Permissive := 1, Comment := 1);   // FV-15-05-01 DIVERT TO SCRAP OR TO DRAIN VALVE
   FV230001_AOI : QSI_Flow_Valve := (DO_Energize := 1, DI_Closed_Feedback := 1, MM_Enable := 1, Config_Opened_Feedback := 1, Config_Closed_Feedback := 1, Config_MO_ResetOnAlarm := 1, Config_TMR_Alm_Preset_ms := 10000, HMI_Alarmed := 1, HMI_Closed := 1, Energize_Permissive := 1, Energize_Enable := 1, ALM := 1, Comment := 1);   // FV-23-00-01 LAUNCH PIG VALVE V1
   FV230002_AOI : QSI_Flow_Valve := (DO_Energize := 1, DI_Closed_Feedback := 1, MM_Enable := 1, Config_Opened_Feedback := 1, Config_Closed_Feedback := 1, Config_MO_ResetOnAlarm := 1, Config_TMR_Alm_Preset_ms := 10000, HMI_Alarmed := 1, HMI_Closed := 1, Energize_Permissive := 1, Energize_Enable := 1, ALM := 1, Comment := 1);   // FV-23-00-02 LAUNCH PIG VALVE V2
   FV2300031_AOI : QSI_Flow_Valve := (DO_Energize := 1, MM_Enable := 1, Config_Opened_Feedback := 1, Config_MO_ResetOnAlarm := 1, Config_TMR_Alm_Preset_ms := 10000, HMI_Alarmed := 1, Energize_Permissive := 1, Energize_Enable := 1, ALM := 1, Comment := 1);   // FV-23-00-03_1 MOVE PIG BACKWARDS INTO CIP/PRODUCTION POSITION
   FV2300032_AOI : QSI_Flow_Valve := (DO_Energize := 1, MM_Enable := 1, Config_Opened_Feedback := 1, Config_MO_ResetOnAlarm := 1, Config_TMR_Alm_Preset_ms := 10000, HMI_Alarmed := 1, Energize_Permissive := 1, Energize_Enable := 1, ALM := 1, Comment := 1);   // FV-23-00-03_2 MOVE PIG FORWARD INTO LAUNCHING POSITION
   FV230004_AOI : QSI_Flow_Valve := (DO_Energize := 1, DI_Closed_Feedback := 1, MM_Enable := 1, Config_Opened_Feedback := 1, Config_Closed_Feedback := 1, Config_MO_ResetOnAlarm := 1, Config_TMR_Alm_Preset_ms := 10000, HMI_Alarmed := 1, HMI_Closed := 1, Energize_Permissive := 1, Energize_Enable := 1, ALM := 1, Comment := 1);   // FV-23-00-04 PIG RETENTION CYLINDER V4.1
   FV230005_AOI : QSI_Flow_Valve := (DO_Energize := 1, DI_Closed_Feedback := 1, MM_Enable := 1, Config_Opened_Feedback := 1, Config_Closed_Feedback := 1, Config_MO_ResetOnAlarm := 1, Config_TMR_Alm_Preset_ms := 10000, HMI_Alarmed := 1, HMI_Closed := 1, Energize_Permissive := 1, Energize_Enable := 1, ALM := 1, Comment := 1);   // FV-23-00-05 PIG RETENTION CYLINDER V4.2
   FV230006_AOI : QSI_Flow_Valve := (DI_Closed_Feedback := 1, MM_Enable := 1, Config_Opened_Feedback := 1, Config_Closed_Feedback := 1, Config_MO_ResetOnAlarm := 1, Config_TMR_Alm_Preset_ms := 10000, HMI_MM := 1, HMI_Closed := 1, Energize_Permissive := 1, Energize_Enable := 1, Comment := 1);   // FV-23-00-06 RETURN PIG TO LAUNCHER VALVE V7
   FV230007_AOI : QSI_Flow_Valve := (DI_Closed_Feedback := 1, MM_Enable := 1, Config_Opened_Feedback := 1, Config_Closed_Feedback := 1, Config_MO_ResetOnAlarm := 1, Config_TMR_Alm_Preset_ms := 10000, HMI_MM := 1, HMI_Closed := 1, Energize_Permissive := 1, Energize_Enable := 1, Comment := 1);   // FV-23-00-07 RETURN PIG TO LAUNCHER VALVE V6
   FV230010_AOI : QSI_Flow_Valve := (DI_Closed_Feedback := 1, MM_Enable := 1, Config_Opened_Feedback := 1, Config_Closed_Feedback := 1, Config_MO_ResetOnAlarm := 1, Config_TMR_Alm_Preset_ms := 10000, HMI_MM := 1, HMI_Alarmed := 1, HMI_Closed := 1, Energize_Permissive := 1, USL_Permissive := 1, LSL_Permissive := 1, Energize_Enable := 1, USL_Enable := 1, LSL_Enable := 1, ALM := 1, Comment := 1);   // FV-23-00-10-O RECEIVING PUMP #1 TO SUCROSE VALVE MANIFOLD MIX PROOF VALVE OPEN
   FV230020_AOI : QSI_Flow_Valve := (DI_Closed_Feedback := 1, MM_Enable := 1, Config_Opened_Feedback := 1, Config_Closed_Feedback := 1, Config_MO_ResetOnAlarm := 1, Config_TMR_Alm_Preset_ms := 10000, HMI_MM := 1, HMI_Alarmed := 1, HMI_Closed := 1, Energize_Permissive := 1, USL_Permissive := 1, LSL_Permissive := 1, Energize_Enable := 1, USL_Enable := 1, LSL_Enable := 1, ALM := 1, Comment := 1);   // FV-23-00-20-O RECEIVING PUMP #2 TO SUCROSE VALVE MANIFOLD MIX PROOF VALVE OPEN
   FV230101_AOI : QSI_Flow_Valve := (DI_Closed_Feedback := 1, MM_Enable := 1, Config_Opened_Feedback := 1, Config_Closed_Feedback := 1, Config_MO_ResetOnAlarm := 1, Config_TMR_Alm_Preset_ms := 10000, HMI_MM := 1, HMI_Closed := 1, Energize_Permissive := 1, USL_Permissive := 1, LSL_Permissive := 1, Comment := 1);   // FV-23-01-01-O SUCROSE RECEIVING TO SUCROSE TANK #1 VALVE OPEN
   FV230102_AOI : QSI_Flow_Valve := (DO_Energize := 1, MM_Enable := 1, Config_MO_ResetOnAlarm := 1, Config_TMR_Alm_Preset_ms := 10000, HMI_MM := 1, HMI_MO := 1, HMI_Opened := 1, Energize_Permissive := 1, Comment := 1);   // FV-23-01-02 SUCROSE TANK #1 INLET/SPRAYBALL VALVE
   FV230103_AOI : QSI_Flow_Valve := (MM_Enable := 1, Config_MO_ResetOnAlarm := 1, Config_TMR_Alm_Preset_ms := 10000, HMI_MO := 1, HMI_Closed := 1, Energize_Permissive := 1, Comment := 1);   // FV-23-01-03 SUCROSE TANK #1 OUTLET VALVE
   FV230104_AOI : QSI_Flow_Valve := (DI_Closed_Feedback := 1, MM_Enable := 1, Config_Opened_Feedback := 1, Config_Closed_Feedback := 1, Config_MO_ResetOnAlarm := 1, Config_TMR_Alm_Preset_ms := 10000, HMI_MM := 1, HMI_Closed := 1, Energize_Permissive := 1, USL_Permissive := 1, LSL_Permissive := 1, Comment := 1);   // FV-23-01-04-O SUCROSE RETURN TO SUCROSE TANK #1 VALVE OPEN
   FV230201_AOI : QSI_Flow_Valve := (DI_Closed_Feedback := 1, MM_Enable := 1, Config_Opened_Feedback := 1, Config_Closed_Feedback := 1, Config_MO_ResetOnAlarm := 1, Config_TMR_Alm_Preset_ms := 10000, HMI_MM := 1, HMI_Closed := 1, Energize_Permissive := 1, USL_Permissive := 1, LSL_Permissive := 1, Comment := 1);   // FV-23-02-01-O SUCROSE RECEIVING TO SUCROSE TANK #2 VALVE OPEN
   FV230202_AOI : QSI_Flow_Valve := (DO_Energize := 1, MM_Enable := 1, Config_MO_ResetOnAlarm := 1, Config_TMR_Alm_Preset_ms := 10000, HMI_MM := 1, HMI_MO := 1, HMI_Opened := 1, Energize_Permissive := 1, Energize_Enable := 1, Comment := 1);   // FV-23-02-02 SUCROSE TANK #2 INLET/SPRAYBALL VALVE
   FV230203_AOI : QSI_Flow_Valve := (MM_Enable := 1, Config_MO_ResetOnAlarm := 1, Config_TMR_Alm_Preset_ms := 10000, HMI_Closed := 1, Energize_Permissive := 1, Comment := 1);   // FV-23-02-03 SUCROSE TANK #2 OUTLET VALVE
   FV230204_AOI : QSI_Flow_Valve := (DI_Closed_Feedback := 1, MM_Enable := 1, Config_Opened_Feedback := 1, Config_Closed_Feedback := 1, Config_MO_ResetOnAlarm := 1, Config_TMR_Alm_Preset_ms := 10000, HMI_MM := 1, HMI_Closed := 1, Energize_Permissive := 1, USL_Permissive := 1, LSL_Permissive := 1, Comment := 1);   // FV-23-02-04-O SUCROSE RETURN TO SUCROSE TANK #2 VALVE OPEN
   FV230222_AOI : QSI_Flow_Valve := (DI_Closed_Feedback := 1, MM_Enable := 1, Config_Opened_Feedback := 1, Config_Closed_Feedback := 1, Config_MO_ResetOnAlarm := 1, Config_TMR_Alm_Preset_ms := 10000, HMI_Alarmed := 1, HMI_Closed := 1, Energize_Permissive := 1, USL_Permissive := 1, LSL_Permissive := 1, ALM := 1, Comment := 1);   // FV-23-02-22-O SUCROSE TANK #2 TO TRANSFER PUMP #2 MIX PROOF VALVE OPEN
   FV230301_AOI : QSI_Flow_Valve := (DI_Closed_Feedback := 1, MM_Enable := 1, Config_Opened_Feedback := 1, Config_Closed_Feedback := 1, Config_MO_ResetOnAlarm := 1, Config_TMR_Alm_Preset_ms := 10000, HMI_MM := 1, HMI_Closed := 1, Energize_Permissive := 1, USL_Permissive := 1, LSL_Permissive := 1, Comment := 1);   // FV-23-03-01-O SUCROSE RECEIVING TO SUCROSE TANK #3 VALVE OPEN
   FV230302_AOI : QSI_Flow_Valve := (DO_Energize := 1, MM_Enable := 1, Config_MO_ResetOnAlarm := 1, Config_TMR_Alm_Preset_ms := 10000, HMI_Opened := 1, Energize_Permissive := 1, Energize_Enable := 1, Comment := 1);   // FV-23-03-02 SUCROSE TANK #3 INLET/SPRAYBALL VALVE
   FV230303_AOI : QSI_Flow_Valve := (MM_Enable := 1, Config_MO_ResetOnAlarm := 1, Config_TMR_Alm_Preset_ms := 10000, HMI_Closed := 1, Energize_Permissive := 1, Comment := 1);   // FV-23-03-03 SUCROSE TANK #3 OUTLET VALVE
   FV230304_AOI : QSI_Flow_Valve := (DI_Closed_Feedback := 1, MM_Enable := 1, Config_Opened_Feedback := 1, Config_Closed_Feedback := 1, Config_MO_ResetOnAlarm := 1, Config_TMR_Alm_Preset_ms := 10000, HMI_MM := 1, HMI_Closed := 1, Energize_Permissive := 1, USL_Permissive := 1, LSL_Permissive := 1, Comment := 1);   // FV-23-03-04-O SUCROSE RETURN TO SUCROSE TANK #3 VALVE OPEN
   FV230401_AOI : QSI_Flow_Valve := (DO_Energize := 1, MM_Enable := 1, Config_MO_ResetOnAlarm := 1, HMI_Opened := 1, Energize_Permissive := 1, Energize_Enable := 1, Comment := 1);   // FV-23-04-01 SUCROSE TANK #3 LOW POINT DRAIN
   FV230402_AOI : QSI_Flow_Valve := (DO_Energize := 1, MM_Enable := 1, Config_MO_ResetOnAlarm := 1, HMI_Opened := 1, Energize_Permissive := 1, Energize_Enable := 1, Comment := 1);   // FV-23-04-02 SUCROSE TANK #2 LOW POINT DRAIN
   FV230403_AOI : QSI_Flow_Valve := (DO_Energize := 1, MM_Enable := 1, Config_MO_ResetOnAlarm := 1, HMI_Opened := 1, Energize_Permissive := 1, Energize_Enable := 1, Comment := 1);   // FV-23-04-03 SUCROSE TANK #1 LOW POINT DRAIN
   FV230411_AOI : QSI_Flow_Valve := (DI_Closed_Feedback := 1, MM_Enable := 1, Config_Opened_Feedback := 1, Config_Closed_Feedback := 1, Config_MO_ResetOnAlarm := 1, Config_TMR_Alm_Preset_ms := 10000, HMI_Alarmed := 1, HMI_Closed := 1, Energize_Permissive := 1, USL_Permissive := 1, LSL_Permissive := 1, ALM := 1, Comment := 1);   // FV-23-04-11-O SUCROSE TANK #1 TO TRANSFER PUMP #1 MIX PROOF VALVE OPEN
   FV230412_AOI : QSI_Flow_Valve := (DI_Closed_Feedback := 1, MM_Enable := 1, Config_Opened_Feedback := 1, Config_Closed_Feedback := 1, Config_MO_ResetOnAlarm := 1, Config_TMR_Alm_Preset_ms := 10000, HMI_Alarmed := 1, HMI_Closed := 1, Energize_Permissive := 1, USL_Permissive := 1, LSL_Permissive := 1, ALM := 1, Comment := 1);   // FV-23-04-12-O SUCROSE TANK #2 TO TRANSFER PUMP #1 MIX PROOF VALVE OPEN
   FV230413_AOI : QSI_Flow_Valve := (DI_Closed_Feedback := 1, MM_Enable := 1, Config_Opened_Feedback := 1, Config_Closed_Feedback := 1, Config_MO_ResetOnAlarm := 1, Config_TMR_Alm_Preset_ms := 10000, HMI_Alarmed := 1, HMI_Closed := 1, Energize_Permissive := 1, USL_Permissive := 1, LSL_Permissive := 1, ALM := 1, Comment := 1);   // FV-23-04-13-O SUCROSE TANK #3 TO TRANSFER PUMP #1 MIX PROOF VALVE OPEN
   FV230421_AOI : QSI_Flow_Valve := (DI_Closed_Feedback := 1, MM_Enable := 1, Config_Opened_Feedback := 1, Config_Closed_Feedback := 1, Config_MO_ResetOnAlarm := 1, Config_TMR_Alm_Preset_ms := 10000, HMI_Alarmed := 1, HMI_Closed := 1, Energize_Permissive := 1, USL_Permissive := 1, LSL_Permissive := 1, ALM := 1, Comment := 1);   // FV-23-04-21-O SUCROSE TANK #1 TO TRANSFER PUMP #2 MIX PROOF VALVE OPEN
   FV230423_AOI : QSI_Flow_Valve := (DI_Closed_Feedback := 1, MM_Enable := 1, Config_Opened_Feedback := 1, Config_Closed_Feedback := 1, Config_MO_ResetOnAlarm := 1, Config_TMR_Alm_Preset_ms := 10000, HMI_Alarmed := 1, HMI_Closed := 1, Energize_Permissive := 1, USL_Permissive := 1, LSL_Permissive := 1, ALM := 1, Comment := 1);   // FV-23-04-23-O SUCROSE TANK #3 TO TRANSFER PUMP #2 MIX PROOF VALVE OPEN
   FV230431_AOI : QSI_Flow_Valve := (DO_Energize := 1, MM_Enable := 1, Config_MO_ResetOnAlarm := 1, HMI_Opened := 1, Energize_Permissive := 1, Energize_Enable := 1, Comment := 1);   // FV-23-04-31 SUCROSE LOW POINT DRAIN VALVE @ TRANSFER PUMP #1
   FV230432_AOI : QSI_Flow_Valve := (DO_Energize := 1, MM_Enable := 1, Config_MO_ResetOnAlarm := 1, HMI_Opened := 1, Energize_Permissive := 1, Energize_Enable := 1, Comment := 1);   // FV-23-04-32 SUCROSE LOW POINT DRAIN VALVE @ TRANSFER PUMP #2
   FV230441_AOI : QSI_Flow_Valve := (DI_Closed_Feedback := 1, MM_Enable := 1, Config_Opened_Feedback := 1, Config_Closed_Feedback := 1, Config_MO_ResetOnAlarm := 1, Config_TMR_Alm_Preset_ms := 10000, HMI_Alarmed := 1, HMI_Closed := 1, Energize_Permissive := 1, USL_Permissive := 1, LSL_Permissive := 1, ALM := 1, Comment := 1);   // FV-23-04-41-O SUCROSE TRANSFER PUMP #1 DISCHARGE TO FILTRATRION MIX PROOF VALVE OPEN
   FV230442_AOI : QSI_Flow_Valve := (DI_Closed_Feedback := 1, MM_Enable := 1, Config_Opened_Feedback := 1, Config_Closed_Feedback := 1, Config_MO_ResetOnAlarm := 1, Config_TMR_Alm_Preset_ms := 10000, HMI_Alarmed := 1, HMI_Closed := 1, Energize_Permissive := 1, USL_Permissive := 1, LSL_Permissive := 1, ALM := 1, Comment := 1);   // FV-23-04-42-O SUCROSE TRANSFER PUMP #2 DISCHARGE TO FILTRATRION MIX PROOF VALVE OPEN
   FV230500_AOI : QSI_Flow_Valve := (MM_Enable := 1, Config_MO_ResetOnAlarm := 1, Config_TMR_Alm_Preset_ms := 10000, HMI_Closed := 1, Energize_Permissive := 1, Comment := 1);   // FV-23-05-00 SUCROSE LOW POINT DRAIN VALVE
   FV230501_AOI : QSI_Flow_Valve := (MM_Enable := 1, Config_Opened_Feedback := 1, Config_Closed_Feedback := 1, Config_MO_ResetOnAlarm := 1, Config_TMR_Alm_Preset_ms := 10000, HMI_Alarmed := 1, Energize_Permissive := 1, USL_Permissive := 1, LSL_Permissive := 1, ALM := 1, Comment := 1);   // FV-23-05-01-O PRE FILTER TRAIN 1 INLET VALVE OPEN
   FV230502_AOI : QSI_Flow_Valve := (MM_Enable := 1, Config_MO_ResetOnAlarm := 1, Config_TMR_Alm_Preset_ms := 10000, HMI_Closed := 1, Energize_Permissive := 1, Comment := 1);   // FV-23-05-02 PRE FILTER TRAIN 1 INLET LOW POINT DRAIN VALVE
   FV230503_AOI : QSI_Flow_Valve := (MM_Enable := 1, Config_MO_ResetOnAlarm := 1, Config_TMR_Alm_Preset_ms := 10000, HMI_Closed := 1, Energize_Permissive := 1, Comment := 1);   // FV-23-05-03 PRE FILTER TRAIN 1 INLET LOW POINT DRAIN VALVE
   FV230504_AOI : QSI_Flow_Valve := (MM_Enable := 1, Config_MO_ResetOnAlarm := 1, Config_TMR_Alm_Preset_ms := 10000, HMI_Closed := 1, Energize_Permissive := 1, Comment := 1);   // FV-23-05-04 PRE FILTER TRAIN 1 OUTLET LOW POINT DRAIN VALVE
   FV230505_AOI : QSI_Flow_Valve := (MM_Enable := 1, Config_MO_ResetOnAlarm := 1, Config_TMR_Alm_Preset_ms := 10000, HMI_Closed := 1, Energize_Permissive := 1, Comment := 1);   // FV-23-05-05 PRE FILTER TRAIN 1 OUTLET LOW POINT DRAIN VALVE
   FV230506_AOI : QSI_Flow_Valve := (MM_Enable := 1, Config_Opened_Feedback := 1, Config_Closed_Feedback := 1, Config_MO_ResetOnAlarm := 1, Config_TMR_Alm_Preset_ms := 10000, HMI_Alarmed := 1, Energize_Permissive := 1, USL_Permissive := 1, LSL_Permissive := 1, ALM := 1, Comment := 1);   // FV-23-05-06-O PRE FILTER TRAIN 1 OUTLET VALVE OPEN
   FV230508_AOI : QSI_Flow_Valve := (MM_Enable := 1, Config_Opened_Feedback := 1, Config_Closed_Feedback := 1, Config_MO_ResetOnAlarm := 1, Config_TMR_Alm_Preset_ms := 10000, HMI_Alarmed := 1, Energize_Permissive := 1, USL_Permissive := 1, LSL_Permissive := 1, ALM := 1, Comment := 1);   // FV-23-05-08-O FINAL FILTER TRAIN 1 INLET VALVE OPEN
   FV230509_AOI : QSI_Flow_Valve := (MM_Enable := 1, Config_MO_ResetOnAlarm := 1, Config_TMR_Alm_Preset_ms := 10000, HMI_Closed := 1, Energize_Permissive := 1, Comment := 1);   // FV-23-05-09 FINAL FILTER TRAIN 1 INLET LOW POINT DRAIN VALVE
   FV230510_AOI : QSI_Flow_Valve := (MM_Enable := 1, Config_MO_ResetOnAlarm := 1, Config_TMR_Alm_Preset_ms := 10000, HMI_Closed := 1, Energize_Permissive := 1, Comment := 1);   // FV-23-05-10 FINAL FILTER TRAIN 1 INLET LOW POINT DRAIN VALVE
   FV230511_AOI : QSI_Flow_Valve := (MM_Enable := 1, Config_MO_ResetOnAlarm := 1, Config_TMR_Alm_Preset_ms := 10000, HMI_Closed := 1, Energize_Permissive := 1, Comment := 1);   // FV-23-05-11 FINAL FILTER TRAIN 1 OUTLET LOW POINT DRAIN VALVE
   FV230512_AOI : QSI_Flow_Valve := (MM_Enable := 1, Config_MO_ResetOnAlarm := 1, Config_TMR_Alm_Preset_ms := 10000, HMI_Closed := 1, Energize_Permissive := 1, Comment := 1);   // FV-23-05-12 FINAL FILTER TRAIN 1 OUTLET LOW POINT DRAIN VALVE
   FV230513_AOI : QSI_Flow_Valve := (MM_Enable := 1, Config_Opened_Feedback := 1, Config_Closed_Feedback := 1, Config_MO_ResetOnAlarm := 1, Config_TMR_Alm_Preset_ms := 10000, HMI_Alarmed := 1, Energize_Permissive := 1, USL_Permissive := 1, LSL_Permissive := 1, ALM := 1, Comment := 1);   // FV-23-05-13-O FINAL FILTER TRAIN 1 OUTLET VALVE OPEN
   FV230601_AOI : QSI_Flow_Valve := (MM_Enable := 1, Config_Opened_Feedback := 1, Config_Closed_Feedback := 1, Config_MO_ResetOnAlarm := 1, Config_TMR_Alm_Preset_ms := 10000, HMI_Alarmed := 1, Energize_Permissive := 1, USL_Permissive := 1, LSL_Permissive := 1, ALM := 1, Comment := 1);   // FV-23-06-01-O PRE FILTER TRAIN 2 INLET VALVE OPEN
   FV230602_AOI : QSI_Flow_Valve := (MM_Enable := 1, Config_MO_ResetOnAlarm := 1, Config_TMR_Alm_Preset_ms := 10000, HMI_Closed := 1, Energize_Permissive := 1, Comment := 1);   // FV-23-06-02 PRE FILTER TRAIN 2 INLET LOW POINT DRAIN VALVE
   FV230603_AOI : QSI_Flow_Valve := (MM_Enable := 1, Config_MO_ResetOnAlarm := 1, Config_TMR_Alm_Preset_ms := 10000, HMI_Closed := 1, Energize_Enable := 1, Comment := 1);   // FV-23-06-03 PRE FILTER TRAIN 2 INLET LOW POINT DRAIN VALVE
   FV230604_AOI : QSI_Flow_Valve := (MM_Enable := 1, Config_MO_ResetOnAlarm := 1, Config_TMR_Alm_Preset_ms := 10000, HMI_Closed := 1, Energize_Permissive := 1, Comment := 1);   // FV-23-06-04 PRE FILTER TRAIN 2 OUTLET LOW POINT DRAIN VALVE
   FV230605_AOI : QSI_Flow_Valve := (MM_Enable := 1, Config_MO_ResetOnAlarm := 1, Config_TMR_Alm_Preset_ms := 10000, HMI_Closed := 1, Energize_Permissive := 1, Comment := 1);   // FV-23-06-05 PRE FILTER TRAIN 2 OUTLET LOW POINT DRAIN VALVE
   FV230606_AOI : QSI_Flow_Valve := (MM_Enable := 1, Config_Opened_Feedback := 1, Config_Closed_Feedback := 1, Config_MO_ResetOnAlarm := 1, Config_TMR_Alm_Preset_ms := 10000, HMI_Alarmed := 1, Energize_Permissive := 1, USL_Permissive := 1, LSL_Permissive := 1, ALM := 1, Comment := 1);   // FV-23-06-06-O PRE FILTER TRAIN 2 OUTLET VALVE OPEN
   FV230607_AOI : QSI_Flow_Valve := (MM_Enable := 1, Config_MO_ResetOnAlarm := 1, Config_TMR_Alm_Preset_ms := 10000, HMI_Closed := 1, Energize_Permissive := 1, Comment := 1);   // FV-23-06-07 LOW POINT DRAIN VALVE
   FV230608_AOI : QSI_Flow_Valve := (MM_Enable := 1, Config_Opened_Feedback := 1, Config_Closed_Feedback := 1, Config_MO_ResetOnAlarm := 1, Config_TMR_Alm_Preset_ms := 10000, HMI_Alarmed := 1, Energize_Permissive := 1, USL_Permissive := 1, LSL_Permissive := 1, ALM := 1, Comment := 1);   // FV-23-06-08-O FINAL FILTER TRAIN 2 INLET VALVE OPEN
   FV230609_AOI : QSI_Flow_Valve := (MM_Enable := 1, Config_MO_ResetOnAlarm := 1, Config_TMR_Alm_Preset_ms := 10000, HMI_Closed := 1, Energize_Permissive := 1, Comment := 1);   // FV-23-06-09 FINAL FILTER TRAIN 2 INLET LOW POINT DRAIN VALVE
   FV230610_AOI : QSI_Flow_Valve := (MM_Enable := 1, Config_MO_ResetOnAlarm := 1, Config_TMR_Alm_Preset_ms := 10000, HMI_Closed := 1, Energize_Permissive := 1, Comment := 1);   // FV-23-06-10 FINAL FILTER TRAIN 2 INLET LOW POINT DRAIN VALVE
   FV230611_AOI : QSI_Flow_Valve := (MM_Enable := 1, Config_MO_ResetOnAlarm := 1, Config_TMR_Alm_Preset_ms := 10000, HMI_Closed := 1, Energize_Permissive := 1, Comment := 1);   // FV-23-06-11 FINAL FILTER TRAIN 2 OUTLET LOW POINT DRAIN VALVE
   FV230612_AOI : QSI_Flow_Valve := (MM_Enable := 1, Config_MO_ResetOnAlarm := 1, Config_TMR_Alm_Preset_ms := 10000, HMI_Closed := 1, Energize_Permissive := 1, Comment := 1);   // FV-23-06-12 FINAL FILTER TRAIN 2 OUTLET LOW POINT DRAIN VALVE
   FV230613_AOI : QSI_Flow_Valve := (MM_Enable := 1, Config_Opened_Feedback := 1, Config_Closed_Feedback := 1, Config_MO_ResetOnAlarm := 1, Config_TMR_Alm_Preset_ms := 10000, HMI_Alarmed := 1, Energize_Permissive := 1, USL_Permissive := 1, LSL_Permissive := 1, ALM := 1, Comment := 1);   // FV-23-06-13-O FINAL FILTER TRAIN 2 OUTLET VALVE OPEN
   FV610010_AOI : QSI_Flow_Valve := (DO_Energize := 1, MM_Enable := 1, Config_NO_Valve := 1, Config_MO_ResetOnAlarm := 1, Config_TMR_Alm_Preset_ms := 10000, HMI_MO := 1, HMI_Closed := 1, Energize_Permissive := 1, Energize_Enable := 1, Comment := 1);   // CIP SUPPLY TO RECEIVING PUMP #1
   FV610020_AOI : QSI_Flow_Valve := (DO_Energize := 1, MM_Enable := 1, Config_MO_ResetOnAlarm := 1, Config_TMR_Alm_Preset_ms := 10000, HMI_Opened := 1, Energize_Permissive := 1, Energize_Enable := 1, Comment := 1);   // CIP SUPPLY TO RECEIVING PUMP #2
   FV610030_AOI : QSI_Flow_Valve := (DO_Energize := 1, MM_Enable := 1, Config_MO_ResetOnAlarm := 1, Config_TMR_Alm_Preset_ms := 10000, HMI_Opened := 1, Energize_Permissive := 1, Energize_Enable := 1, Comment := 1);   // LOW POINT DRAIN VALVE
   FV610101_AOI : QSI_Flow_Valve := (DI_Closed_Feedback := 1, MM_Enable := 1, Config_Opened_Feedback := 1, Config_Closed_Feedback := 1, Config_MO_ResetOnAlarm := 1, Config_TMR_Alm_Preset_ms := 10000, HMI_MM := 1, HMI_Closed := 1, Energize_Permissive := 1, USL_Permissive := 1, LSL_Permissive := 1, Comment := 1);   // FV-61-01-01-O CIP SUPPLY TO SUCROSE TANK #1 VALVE OPEN
   FV610201_AOI : QSI_Flow_Valve := (DI_Closed_Feedback := 1, MM_Enable := 1, Config_Opened_Feedback := 1, Config_Closed_Feedback := 1, Config_MO_ResetOnAlarm := 1, Config_TMR_Alm_Preset_ms := 10000, HMI_MM := 1, HMI_Closed := 1, Energize_Permissive := 1, USL_Permissive := 1, LSL_Permissive := 1, Energize_Enable := 1, USL_Enable := 1, LSL_Enable := 1, Comment := 1);   // FV-61-02-01-O CIP SUPPLY TO SUCROSE TANK #2 VALVE OPEN
   FV610301_AOI : QSI_Flow_Valve := (DI_Closed_Feedback := 1, MM_Enable := 1, Config_Opened_Feedback := 1, Config_Closed_Feedback := 1, Config_MO_ResetOnAlarm := 1, Config_TMR_Alm_Preset_ms := 10000, HMI_MM := 1, HMI_Closed := 1, Energize_Permissive := 1, USL_Permissive := 1, LSL_Permissive := 1, Comment := 1);   // FV-61-03-01-O CIP SUPPLY TO SUCROSE TANK #3 VALVE OPEN
   FV610401_AOI : QSI_Flow_Valve := (DI_Closed_Feedback := 1, MM_Enable := 1, Config_Opened_Feedback := 1, Config_Closed_Feedback := 1, Config_MO_ResetOnAlarm := 1, Config_TMR_Alm_Preset_ms := 10000, HMI_MM := 1, HMI_Closed := 1, Energize_Permissive := 1, USL_Permissive := 1, LSL_Permissive := 1, Energize_Enable := 1, USL_Enable := 1, LSL_Enable := 1, Comment := 1);   // FV-61-04-01-O VALVE MANIFOLD TO SUCROSE TRANSFER PUMP #1 VALVE OPEN
   FV610402_AOI : QSI_Flow_Valve := (DI_Closed_Feedback := 1, MM_Enable := 1, Config_Opened_Feedback := 1, Config_Closed_Feedback := 1, Config_MO_ResetOnAlarm := 1, Config_TMR_Alm_Preset_ms := 10000, HMI_MM := 1, HMI_Closed := 1, Energize_Permissive := 1, USL_Permissive := 1, LSL_Permissive := 1, Energize_Enable := 1, USL_Enable := 1, LSL_Enable := 1, Comment := 1);   // FV-61-04-02-O VALVE MANIFOLD TO SUCROSE TRANSFER PUMP #2 VALVE OPEN
   FV610411_AOI : QSI_Flow_Valve := (DO_Energize := 1, MM_Enable := 1, Config_MO_ResetOnAlarm := 1, Config_TMR_Alm_Preset_ms := 10000, HMI_Opened := 1, Energize_Permissive := 1, Energize_Enable := 1, Comment := 1);   // FV-61-04-11 CIP SUPPLY TO TRANSFER PUMP #1 OR TO DRAIN DIVERT VALVE
   FV610412_AOI : QSI_Flow_Valve := (DO_Energize := 1, MM_Enable := 1, Config_MO_ResetOnAlarm := 1, Config_TMR_Alm_Preset_ms := 10000, HMI_Opened := 1, Energize_Permissive := 1, Energize_Enable := 1, Comment := 1);   // FV-61-04-12 CIP SUPPLY TO TRANSFER PUMP #2 OR TO DRAIN DIVERT VALVE
   FV610501_AOI : QSI_Flow_Valve := (DI_Closed_Feedback := 1, MM_Enable := 1, Config_Opened_Feedback := 1, Config_Closed_Feedback := 1, Config_MO_ResetOnAlarm := 1, Config_TMR_Alm_Preset_ms := 10000, HMI_Alarmed := 1, HMI_Closed := 1, Energize_Permissive := 1, USL_Permissive := 1, LSL_Permissive := 1, ALM := 1, Comment := 1);   // FV-61-05-01-O CIP SUPPLY TO FILTRATION AND RING MAIN MIX PROOF VALVE OPEN
   FV620010_AOI : QSI_Flow_Valve := (DO_Energize := 1, DO_USL_Energize := 1, DO_LSL_Energize := 1, DI_Closed_Feedback := 1, MM_Enable := 1, Config_Opened_Feedback := 1, Config_Closed_Feedback := 1, Config_MO_ResetOnAlarm := 1, Config_TMR_Alm_Preset_ms := 10000, HMI_Alarmed := 1, HMI_Closed := 1, Energize_Permissive := 1, USL_Permissive := 1, LSL_Permissive := 1, Energize_Enable := 1, USL_Enable := 1, LSL_Enable := 1, ALM := 1, Comment := 1);   // FV-62-00-10-O RECEIVING PUMP #1 TO CIP RETURN MIX PROOF VALVE OPEN
   FV620020_AOI : QSI_Flow_Valve := (DO_Energize := 1, DO_USL_Energize := 1, DO_LSL_Energize := 1, DI_Closed_Feedback := 1, MM_Enable := 1, Config_Opened_Feedback := 1, Config_Closed_Feedback := 1, Config_MO_ResetOnAlarm := 1, Config_TMR_Alm_Preset_ms := 10000, HMI_Alarmed := 1, HMI_Closed := 1, Energize_Permissive := 1, USL_Permissive := 1, LSL_Permissive := 1, Energize_Enable := 1, USL_Enable := 1, LSL_Enable := 1, ALM := 1, Comment := 1);   // FV-62-00-20-O RECEIVING PUMP #2 TO CIP RETURN MIX PROOF VALVE OPEN
   FV620101_AOI : QSI_Flow_Valve := (DI_Closed_Feedback := 1, MM_Enable := 1, Config_Opened_Feedback := 1, Config_Closed_Feedback := 1, Config_MO_ResetOnAlarm := 1, Config_TMR_Alm_Preset_ms := 10000, HMI_Alarmed := 1, HMI_Closed := 1, Energize_Permissive := 1, USL_Permissive := 1, LSL_Permissive := 1, ALM := 1, Comment := 1);   // FV-62-01-01-O SUCROSE TANK #1 TO CIP RETURN PUMP MIX PROOF VALVE OPEN
   FV620201_AOI : QSI_Flow_Valve := (DO_Energize := 1, DI_Closed_Feedback := 1, MM_Enable := 1, Config_Opened_Feedback := 1, Config_Closed_Feedback := 1, Config_MO_ResetOnAlarm := 1, Config_TMR_Alm_Preset_ms := 10000, HMI_Alarmed := 1, HMI_Closed := 1, Energize_Permissive := 1, USL_Permissive := 1, LSL_Permissive := 1, Energize_Enable := 1, ALM := 1, Comment := 1);   // FV-62-02-01-O SUCROSE TANK #2 TO CIP RETURN PUMP MIX PROOF VALVE OPEN
   FV620301_AOI : QSI_Flow_Valve := (DO_Energize := 1, DI_Closed_Feedback := 1, MM_Enable := 1, Config_Opened_Feedback := 1, Config_Closed_Feedback := 1, Config_MO_ResetOnAlarm := 1, Config_TMR_Alm_Preset_ms := 10000, HMI_Alarmed := 1, HMI_Closed := 1, Energize_Permissive := 1, USL_Permissive := 1, LSL_Permissive := 1, Energize_Enable := 1, ALM := 1, Comment := 1);   // FV-62-03-01-O SUCROSE TANK #3 TO CIP RETURN PUMP MIX PROOF VALVE OPEN
   FV620400_AOI : QSI_Flow_Valve := (MM_Enable := 1, Config_MO_ResetOnAlarm := 1, Config_TMR_Alm_Preset_ms := 10000, HMI_Closed := 1, Energize_Permissive := 1, Comment := 1);   // FV-62-04-00 CIP RETURN LOW POINT DRAIN VALVE
   FV620401_AOI : QSI_Flow_Valve := (DI_Closed_Feedback := 1, MM_Enable := 1, Config_Opened_Feedback := 1, Config_Closed_Feedback := 1, Config_MO_ResetOnAlarm := 1, Config_TMR_Alm_Preset_ms := 10000, HMI_Alarmed := 1, HMI_Closed := 1, Energize_Permissive := 1, USL_Permissive := 1, LSL_Permissive := 1, ALM := 1, Comment := 1);   // FV-62-04-01-O CIP RETURN PUMP #1 TO FILTER SYSTEM MIX PROOF VALVE OPEN
   FV620402_AOI : QSI_Flow_Valve := (DI_Closed_Feedback := 1, MM_Enable := 1, Config_Opened_Feedback := 1, Config_Closed_Feedback := 1, Config_MO_ResetOnAlarm := 1, Config_TMR_Alm_Preset_ms := 10000, HMI_Alarmed := 1, HMI_Closed := 1, Energize_Permissive := 1, USL_Permissive := 1, LSL_Permissive := 1, ALM := 1, Comment := 1);   // FV-62-04-02-O CIP RETURN PUMP #2 TO FILTER SYSTEM MIX PROOF VALVE OPEN
   FV620701_AOI : QSI_Flow_Valve := (DI_Closed_Feedback := 1, MM_Enable := 1, Config_Opened_Feedback := 1, Config_Closed_Feedback := 1, Config_MO_ResetOnAlarm := 1, Config_TMR_Alm_Preset_ms := 10000, HMI_MM := 1, HMI_Closed := 1, Energize_Permissive := 1, USL_Permissive := 1, LSL_Permissive := 1, Comment := 1);   // FV-62-07-01-O SUCROSE RING MAIN RETURN TO CIP RETURN VALVE VALVE OPEN
   FV621001_AOI : QSI_Flow_Valve := (DI_Closed_Feedback := 1, MM_Enable := 1, Config_Opened_Feedback := 1, Config_Closed_Feedback := 1, Config_MO_ResetOnAlarm := 1, Config_TMR_Alm_Preset_ms := 10000, HMI_MM := 1, HMI_Closed := 1, Energize_Permissive := 1, USL_Permissive := 1, LSL_Permissive := 1, Energize_Enable := 1, Comment := 1);   // FV-62-10-01-O SUCROSE RECEIVING TO CIP RETURN VALVE OPEN
   FV740301_AOI : QSI_Flow_Valve := (MM_Enable := 1, Config_MO_ResetOnAlarm := 1, Config_TMR_Alm_Preset_ms := 10000, HMI_MM := 1, HMI_Closed := 1, Energize_Permissive := 1, Energize_Enable := 1, Comment := 1);   // FV-74-03-01 STEAM SIP SUPPLY VALVE
   FV740401_AOI : QSI_Flow_Valve := (MM_Enable := 1, Config_MO_ResetOnAlarm := 1, Config_TMR_Alm_Preset_ms := 10000, HMI_Closed := 1, Energize_Permissive := 1, Comment := 1);   // FV-74-04-01 SIP SUPPLY VALVE
   FV740501_AOI : QSI_Flow_Valve := (MM_Enable := 1, Config_MO_ResetOnAlarm := 1, Config_TMR_Alm_Preset_ms := 10000, HMI_Closed := 1, Energize_Permissive := 1, Comment := 1);   // FV-74-05-01 SIP SUPPLY TO PRE FILTER TRAIN 1 VALVE
   FV740502_AOI : QSI_Flow_Valve := (MM_Enable := 1, Config_MO_ResetOnAlarm := 1, Config_TMR_Alm_Preset_ms := 10000, HMI_Closed := 1, Energize_Permissive := 1, Comment := 1);   // FV-74-05-02 SIP SUPPLY TO FINAL FILTER TRAIN 1 VALVE
   FV740601_AOI : QSI_Flow_Valve := (MM_Enable := 1, Config_MO_ResetOnAlarm := 1, Config_TMR_Alm_Preset_ms := 10000, HMI_Closed := 1, Energize_Permissive := 1, Comment := 1);   // FV-74-06-01 SIP SUPPLY TO PRE FILTER TRAIN 2 VALVE
   FV740602_AOI : QSI_Flow_Valve := (MM_Enable := 1, Config_MO_ResetOnAlarm := 1, Config_TMR_Alm_Preset_ms := 10000, HMI_Closed := 1, Energize_Permissive := 1, Comment := 1);   // FV-74-06-02 SIP SUPPLY TO FINAL FILTER TRAIN 2 VALVE
   FV750501_AOI : QSI_Flow_Valve := (MM_Enable := 1, Config_MO_ResetOnAlarm := 1, Config_TMR_Alm_Preset_ms := 10000, HMI_Closed := 1, Energize_Permissive := 1, Comment := 1);   // FV-75-05-01 TRP-75-05-01 ISOLATION VALVE
   FV750502_AOI : QSI_Flow_Valve := (MM_Enable := 1, Config_MO_ResetOnAlarm := 1, Config_TMR_Alm_Preset_ms := 10000, HMI_Closed := 1, Energize_Permissive := 1, Comment := 1);   // FV-75-05-02 TRP-75-05-02 ISOLATION VALVE
   FV750503_AOI : QSI_Flow_Valve := (MM_Enable := 1, Config_MO_ResetOnAlarm := 1, Config_TMR_Alm_Preset_ms := 10000, HMI_Closed := 1, Energize_Permissive := 1, Comment := 1);   // FV-75-05-03 TRP-75-05-03 ISOLATION VALVE
   FV750504_AOI : QSI_Flow_Valve := (MM_Enable := 1, Config_MO_ResetOnAlarm := 1, Config_TMR_Alm_Preset_ms := 10000, HMI_Closed := 1, Energize_Permissive := 1, Comment := 1);   // FV-75-05-04 TRP-75-05-04 ISOLATION VALVE
   FV750601_AOI : QSI_Flow_Valve := (MM_Enable := 1, Config_MO_ResetOnAlarm := 1, Config_TMR_Alm_Preset_ms := 10000, HMI_Closed := 1, Energize_Permissive := 1, Comment := 1);   // FV-75-06-01 TRP-75-06-01 ISOLATION VALVE
   FV750602_AOI : QSI_Flow_Valve := (MM_Enable := 1, Config_MO_ResetOnAlarm := 1, HMI_Closed := 1, Energize_Permissive := 1, Comment := 1);   // FV-75-06-02 TRP-75-06-02 ISOLATION VALVE
   FV750603_AOI : QSI_Flow_Valve := (MM_Enable := 1, Config_MO_ResetOnAlarm := 1, Config_TMR_Alm_Preset_ms := 10000, HMI_Closed := 1, Energize_Permissive := 1, Comment := 1);   // FV-75-06-03 TRP-75-06-03 ISOLATION VALVE
   FV750604_AOI : QSI_Flow_Valve := (MM_Enable := 1, Config_MO_ResetOnAlarm := 1, Config_TMR_Alm_Preset_ms := 10000, HMI_Closed := 1, Energize_Permissive := 1, Comment := 1);   // FV-75-06-04 TRP-75-06-04 ISOLATION VALVE
   FV751101_AOI : QSI_Flow_Valve := (MM_Enable := 1, Config_MO_ResetOnAlarm := 1, Config_TMR_Alm_Preset_ms := 10000, HMI_Closed := 1, Energize_Permissive := 1, Comment := 1);   // FV-75-11-01 SUCROSE TANK #1 BLANKETING STEAM TRAP ISOLATION VALVE
   FV751201_AOI : QSI_Flow_Valve := (DO_Energize := 1, MM_Enable := 1, Config_MO_ResetOnAlarm := 1, Config_TMR_Alm_Preset_ms := 10000, HMI_Opened := 1, Energize_Permissive := 1, Energize_Enable := 1, Comment := 1);   // FV-75-12-01 SUCROSE TANK #2 BLANKETING STEAM TRAP ISOLATION VALVE
   FV751301_AOI : QSI_Flow_Valve := (DO_Energize := 1, MM_Enable := 1, Config_MO_ResetOnAlarm := 1, Config_TMR_Alm_Preset_ms := 10000, HMI_Opened := 1, Energize_Permissive := 1, Energize_Enable := 1, Comment := 1);   // FV-75-13-01 SUCROSE TANK #3 BLANKETING STEAM TRAP ISOLATION VALVE
   FV751401_AOI : QSI_Flow_Valve := (DO_Energize := 1, MM_Enable := 1, Config_MO_ResetOnAlarm := 1, Config_TMR_Alm_Preset_ms := 10000, HMI_Opened := 1, Energize_Permissive := 1, Energize_Enable := 1, Comment := 1);   // FV-75-14-01 CONDENSATE TANK BLANKETING STEAM TRAP ISOLATION VALVE
   FV920301_AOI : QSI_Flow_Valve := (MM_Enable := 1, Config_NO_Valve := 1, Config_MO_ResetOnAlarm := 1, Config_TMR_Alm_Preset_ms := 10000, HMI_MM := 1, HMI_Opened := 1, Energize_Permissive := 1, Energize_Enable := 1, Comment := 1);   // FV-92-03-01 INSTRUMENT AIR HEATER ISOLATION VALVE
   FV920501_AOI : QSI_Flow_Valve := (MM_Enable := 1, Config_MO_ResetOnAlarm := 1, Config_TMR_Alm_Preset_ms := 10000, HMI_Closed := 1, Energize_Permissive := 1, Comment := 1);   // FV-92-05-01 FLT-23-05-01 VENT VALVE
   FV920502_AOI : QSI_Flow_Valve := (MM_Enable := 1, Config_MO_ResetOnAlarm := 1, Config_TMR_Alm_Preset_ms := 10000, HMI_Closed := 1, Energize_Permissive := 1, Comment := 1);   // FV-92-05-02 FLT-23-05-02 VENT VALVE
   FV920601_AOI : QSI_Flow_Valve := (MM_Enable := 1, Config_MO_ResetOnAlarm := 1, Config_TMR_Alm_Preset_ms := 10000, HMI_Closed := 1, Energize_Permissive := 1, Comment := 1);   // FV-92-06-01 FLT-23-06-01 VENT VALVE
   FV920602_AOI : QSI_Flow_Valve := (MM_Enable := 1, Config_MO_ResetOnAlarm := 1, Config_TMR_Alm_Preset_ms := 10000, HMI_Closed := 1, Energize_Permissive := 1, Comment := 1);   // FV-92-06-02 FLT-23-06-02 VENT VALVE
   FV930401_AOI : QSI_Flow_Valve := (MM_Enable := 1, Config_MO_ResetOnAlarm := 1, Config_TMR_Alm_Preset_ms := 10000, HMI_Closed := 1, Energize_Permissive := 1, Comment := 1);   // FV-93-04-01 FLT-93-04-01 INLET VALVE
   FV930501_AOI : QSI_Flow_Valve := (MM_Enable := 1, Config_MO_ResetOnAlarm := 1, Config_TMR_Alm_Preset_ms := 10000, HMI_Closed := 1, Energize_Permissive := 1, Comment := 1);   // FV-93-05-01 PRE FILTER TRAIN 1 AIR BLOW INLET
   FV930502_AOI : QSI_Flow_Valve := (MM_Enable := 1, Config_MO_ResetOnAlarm := 1, Config_TMR_Alm_Preset_ms := 10000, HMI_Closed := 1, Energize_Permissive := 1, Comment := 1);   // FV-93-05-02 FINAL FILTER TRAIN 1 AIR BLOW VALVE
   FV930503_AOI : QSI_Flow_Valve := (MM_Enable := 1, Config_MO_ResetOnAlarm := 1, Config_TMR_Alm_Preset_ms := 10000, HMI_Closed := 1, Energize_Permissive := 1, Comment := 1);   // FV-93-05-03 INTEGRITY TEST TO SUPPLY TO FINAL FILTER TRAIN 1 VALVE
   FV930511_AOI : QSI_Flow_Valve := (MM_Enable := 1, Config_MO_ResetOnAlarm := 1, Config_TMR_Alm_Preset_ms := 10000, HMI_Closed := 1, Energize_Permissive := 1, Comment := 1);   // FV-93-05-11 PRE FILTER TRAIN 1 AIR BLOW OUTLET
   FV930512_AOI : QSI_Flow_Valve := (MM_Enable := 1, Config_MO_ResetOnAlarm := 1, Config_TMR_Alm_Preset_ms := 10000, HMI_Closed := 1, Energize_Permissive := 1, Comment := 1);   // FV-93-05-12 FINAL FILTER TRAIN 1 AIR BLOW OUTLET
   FV930601_AOI : QSI_Flow_Valve := (MM_Enable := 1, Config_MO_ResetOnAlarm := 1, Config_TMR_Alm_Preset_ms := 10000, HMI_Closed := 1, Energize_Permissive := 1, Comment := 1);   // FV-93-06-01 PRE FILTER TRAIN 2 AIR BLOW INLET
   FV930602_AOI : QSI_Flow_Valve := (MM_Enable := 1, Config_MO_ResetOnAlarm := 1, Config_TMR_Alm_Preset_ms := 10000, HMI_Closed := 1, Energize_Permissive := 1, Comment := 1);   // FV-93-06-02 FINAL FILTER TRAIN 2 AIR BLOW OUTLET
   FV930603_AOI : QSI_Flow_Valve := (MM_Enable := 1, Config_MO_ResetOnAlarm := 1, Config_TMR_Alm_Preset_ms := 10000, HMI_Closed := 1, Energize_Permissive := 1, Comment := 1);   // FV-93-06-03 INTEGRITY TEST TO SUPPLY TO FINAL FILTER DRAIN VALVE
   FV930611_AOI : QSI_Flow_Valve := (MM_Enable := 1, Config_MO_ResetOnAlarm := 1, Config_TMR_Alm_Preset_ms := 10000, HMI_Closed := 1, Energize_Permissive := 1, Comment := 1);   // FV-93-06-11 PRE FILTER TRAIN 2 AIR BLOW OUTLET
   FV930612_AOI : QSI_Flow_Valve := (MM_Enable := 1, Config_MO_ResetOnAlarm := 1, Config_TMR_Alm_Preset_ms := 10000, HMI_Closed := 1, Energize_Permissive := 1, Comment := 1);   // FV-93-06-12 FINAL FILTER TRAIN 2 AIR BLOW OUTLET
   FV931101_AOI : QSI_Flow_Valve := (MM_Enable := 1, Config_MO_ResetOnAlarm := 1, Config_TMR_Alm_Preset_ms := 10000, HMI_Closed := 1, Energize_Permissive := 1, Comment := 1);   // FV-93-11-01 STERILE AIR FLT-93-11-01 SHUT OFF VALVE
   FV931102_AOI : QSI_Flow_Valve := (Config_NO_Valve := 1, Config_MO_ResetOnAlarm := 1);
   FV931103_AOI : QSI_Flow_Valve := (Config_NO_Valve := 1);
   FV931201_AOI : QSI_Flow_Valve := (DO_Energize := 1, MM_Enable := 1, Config_MO_ResetOnAlarm := 1, Config_TMR_Alm_Preset_ms := 10000, HMI_Opened := 1, Energize_Permissive := 1, Energize_Enable := 1, Comment := 1);   // FV-93-12-01 STERILE AIR FLT-93-12-01 SHUT OFF VALVE
   FV931202_AOI : QSI_Flow_Valve := (Config_NO_Valve := 1, Config_MO_ResetOnAlarm := 1);
   FV931203_AOI : QSI_Flow_Valve := (Config_NO_Valve := 1);
   FV931301_AOI : QSI_Flow_Valve := (DO_Energize := 1, MM_Enable := 1, Config_MO_ResetOnAlarm := 1, Config_TMR_Alm_Preset_ms := 10000, HMI_Opened := 1, Energize_Permissive := 1, Energize_Enable := 1, Comment := 1);   // FV-93-13-01 STERILE AIR FLT-93-13-01 SHUT OFF VALVE
   FV931302_AOI : QSI_Flow_Valve := (Config_NO_Valve := 1);
   FV931303_AOI : QSI_Flow_Valve := (Config_NO_Valve := 1);
   HEADER_FLOW_SP : DINT;
   HEADER_LOW_FLOW : DINT;
   HOT_WATER_FLOW : DINT;
   HOT_WATER_TEMP : DINT;
   HRM_SIP250TimeRemaining : DINT;
   HRM_SIP254TimeRemaining : DINT;
   HRM_StepTimeRemaining : DINT;
   HTR760101_AOI : QSI_Discrete_Device := (DO_Energize := 1, MM_Enable := 1, Config_MO_ResetOnAlarm := 1, Config_TMR_Alm_Preset_ms := 10000, HMI_Energized := 1, HMI_Disconnect_OK := 1, Energize_Permissive := 1, Energize_Enable := 1, Comment := 1);   // HTR-76-01-01 SUCROSE TANK #1 UTILITY HOT WATER ELECTRIC HEATER ENABLE
   HTR760201_AOI : QSI_Discrete_Device := (DO_Energize := 1, MM_Enable := 1, Config_MO_ResetOnAlarm := 1, Config_TMR_Alm_Preset_ms := 10000, HMI_Energized := 1, HMI_Disconnect_OK := 1, Energize_Permissive := 1, Energize_Enable := 1, Comment := 1);   // HTR-76-02-01 SUCROSE TANK #2 UTILITY HOT WATER ELECTRIC HEATER ENABLE
   HTR760301_AOI : QSI_Discrete_Device := (DO_Energize := 1, MM_Enable := 1, Config_MO_ResetOnAlarm := 1, Config_TMR_Alm_Preset_ms := 10000, HMI_Energized := 1, HMI_Disconnect_OK := 1, Energize_Permissive := 1, Energize_Enable := 1, Comment := 1);   // HTR-76-03-01 SUCROSE TANK #3 UTILITY HOT WATER ELECTRIC HEATER ENABLE
   HTR920301_AOI : QSI_Discrete_Device := (DO_Energize := 1, MM_Enable := 1, Config_MO_ResetOnAlarm := 1, Config_TMR_Alm_Preset_ms := 10000, HMI_Energized := 1, HMI_Disconnect_OK := 1, Energize_Permissive := 1, Energize_Enable := 1, Comment := 1);   // HTR-92-03-01 COMPRESSED AIR TANK AIR BLANKETING HEATER
   Integrity_Control : CONTROL;
   Integrity_Result : DINT;
   Integrity_Test_FIFO : REAL[15];
   IO_Check : BOOL;
   MAP_TO_SUCROSE_CIP : DINT[10];
        [0].4   // OK TO CIP TANK 2 INTERLOCK
        [0].0   // OK TO CIP RECEIVING 1 SKID INTERLOCK
        [0].1   // OK TO CIP RECEIVING 2 SKID INTERLOCK
        [0].3   // OK TO CIP TANK 1 INTERLOCK
        [0].2   // OK TO CIP RECEIVING AND LINE INTERLOCK
        [0].5   // OK TO CIP TANK 3 INTERLOCK
        [0].6   // OK TO CIP P230401 INTERLOCK
        [0].7   // OK TO CIP P230402 INTERLOCK
        [0].8   // OK TO CIP FILTRATION SKID INTERLOCK
        [0].16   // OK TO SANITIZE TANK 1 INTERLOCK
        [0].17   // OK TO SANITIZE TANK 2 INTERLOCK
        [0].18   // OK TO SANITIZE TANK 3 INTERLOCK
   Messaging : Area_Ladder := (BIT_Alarm[0] := 1, SP_Logic[0] := 2, TMR_Logic[0].EN := 1, TMR_Logic[0].TT := 1, TMR_Logic[9].ACC := 5, TMR_Logic[9].EN := 1, TMR_Logic[9].DN := 1);
   MSG_READ_FROM_CIP3 : MESSAGE;
   MSG_READ_FROM_SUCROSE_CIP : MESSAGE;
        MessageParameters(ServiceCode := 16#004c, LocalElement := READ_FROM_SUCROSE_CIP[0], ...)
   New_Sec : BOOL;
   ONESHOTBITS : INT[10];
   P230010_AOI : PF525_VFD_E_ENET := (MM_Enable := 1, Config_TMR_Alm_Preset := 10000, Config_PID := 1, AS1_Enable := 1, AS2_Enable := 1, HMI_MS := 10, ALM := 1);   // P-23-00-10 RECEIVING PUMP 1
   P230020_AOI : PF525_VFD_E_ENET := (MM_Enable := 1, Config_TMR_Alm_Preset := 10000, HMI_MS := 10);   // P-23-00-20 RECEIVING PUMP 2
   P230401_AOI : PF525_VFD_E_ENET := (MM_Enable := 1, Config_TMR_On_Preset := 10000, Config_TMR_Alm_Preset := 10000, Config_AS1 := 1, SP_AS1 := 25, Start_Permissive := 1, HMI_MM := 1, HMI_MS := 10, ALM := 1);   // P-23-04-01 SUCROSE TRANSFER PUMP 1
   P230402_AOI : PF525_VFD_E_ENET := (MM_Enable := 1, Config_TMR_On_Preset := 10000, Config_TMR_Alm_Preset := 10000, Config_AS1 := 1, SP_AS1 := 25, Start_Permissive := 1, HMI_MM := 1, HMI_MS := 10, ALM := 1);   // P-23-04-02 SUCROSE TRANSFER PUMP 2
   P620101_AOI : PF525_VFD_E_ENET := (MM_Enable := 1, Config_TMR_Alm_Preset := 10000, Config_AS1 := 1, Config_AS2 := 1, SP_AS1 := 95, SP_AS2 := 50, Start_Permissive := 1, HMI_MM := 1, HMI_MS := 10, ALM := 1);   // P-62-01-01 CIP RETURN UP
   PAG : BOOL;   // Test Bit
   PBL1604001_AOI : QSI_Discrete_Device := (DO_Energize := 1, MM_Enable := 1, Config_MO_ResetOnAlarm := 1, HMI_Energized := 1, HMI_Disconnect_OK := 1, Energize_Permissive := 1, Energize_Enable := 1, Comment := 1);   // PBL-16040-01 RESET PB LIGHT
   PBL1604002_AOI : QSI_Discrete_Device := (DO_Energize := 1, MM_Enable := 1, Config_Energized_Text := 1, Config_MO_ResetOnAlarm := 1, Config_TMR_Alm_Preset_ms := 10000, HMI_Energized := 1, HMI_Disconnect_OK := 1, Energize_Permissive := 1, Energize_Enable := 1, Comment := 1);   // PBL-16040-02 E-STOP CIRCUIT RESET LIGHT
   PI_E25_1 : REAL[2];   // Analog Input EN2T_FLX 192.168.1.25
        [0]   // FIT-23-00-10 MASS FLOW METER FOR RECEIVING PUMP P-23-00-10
        [1]   // FIT-23-00-20 MASS FLOW METER FOR RECEIVING PUMP P-23-00-20
   PIT_93_01_01_HIGH_PRESS : DINT;
   PIT_93_01_01_LOW_PRESS : DINT;
   PIT_93_02_01_HIGH_PRESS : DINT;
   PIT_93_02_01_LOW_PRESS : DINT;
   PIT_93_03_01_HIGH_PRESS : DINT;
   PIT_93_03_01_LOW_PRESS : DINT;
   PSV230010_AOI : QSI_Flow_Valve := (DO_Energize := 1, MM_Enable := 1, Config_MO_ResetOnAlarm := 1, Config_TMR_Alm_Preset_ms := 10000, HMI_Opened := 1, Energize_Permissive := 1, Energize_Enable := 1, Comment := 1);
   PSV230010_AOI111 : QSI_Flow_Valve := (Config_Opened_Feedback := 1, Config_Closed_Feedback := 1, Config_MO_ResetOnAlarm := 1);
   PSV230020_AOI : QSI_Flow_Valve := (DO_Energize := 1, MM_Enable := 1, Config_MO_ResetOnAlarm := 1, Config_TMR_Alm_Preset_ms := 10000, HMI_Opened := 1, Energize_Permissive := 1, Energize_Enable := 1, Comment := 1);
   PSV230401_AOI : QSI_Flow_Valve := (MM_Enable := 1, Config_MO_ResetOnAlarm := 1, Config_TMR_Alm_Preset_ms := 10000, HMI_MO := 1, HMI_Closed := 1, Energize_Permissive := 1, Comment := 1);   // PSV-23-04-01 TRANSFER PUMP #1 BYPASS VALVE
   PSV230402_AOI : QSI_Flow_Valve := (MM_Enable := 1, Config_MO_ResetOnAlarm := 1, Config_TMR_Alm_Preset_ms := 10000, HMI_Closed := 1, Energize_Permissive := 1, Comment := 1);   // PSV-23-04-02 TRANSFER PUMP #2 BYPASS VALVE
   READ_FROM_CIP3 : INT[5];
   READ_FROM_SUCROSE_CIP : DINT[10];
        [2]   // HOT WATER TEMP FROM CIP SKID
        [1]   // HOT WATER FLOW FROM CIP SKID
   ReceivingArea : Area_Program;
   Rung_Comment : BOOL := 1;
   SECURITY : User_Login;
   SUCROSE_HEADER_NO_ALARM : BOOL := 1;
   SUCROSE_HEADER_WATER_PURGE_GALLONS_TOTAL : DINT;
   SUCROSE_HEADER_WATER_PURGE_SP : DINT;
   Sucrose_MM_Enable : BOOL := 1;
   SUCROSE_TANK_QUEUE_LEVEL : DINT := 50;
   SucroseCIP_Drain_Inhibit : BOOL;
   SucroseCIP_FILTRATION_ALL_PATHS_Selected : BOOL;
   SucroseCIP_FILTRATION_PATH1_Selected : BOOL;
   SucroseCIP_FILTRATION_PATH2_Selected : BOOL;
   SucroseCIP_FILTRATION_PATH3_Selected : BOOL;
   SucroseCIP_FILTRATION_PATH4_Selected : BOOL;
   SucroseCIP_FILTRATION_REMOTE : CIP_REMOTE;
   SucroseCIP_HELD : BOOL;
   SucroseCIP_P230401_REMOTE : CIP_REMOTE := (BIT_ONS[0] := 1, BIT_ONS[1] := 1);
   SucroseCIP_P230402_REMOTE : CIP_REMOTE := (BIT_ONS[0] := 1, BIT_ONS[1] := 1);
   SucroseCIP_PAUSED : BOOL;
   SucroseCIP_Pulse_Inhibit : BOOL;
   SucroseCIP_RECEIVING2_REMOTE : CIP_REMOTE;
   SucroseCIP_RECEIVING_LINE_REMOTE : CIP_REMOTE;
   SucroseCIP_RECEIVING_REMOTE : CIP_REMOTE := (BIT_ONS[0] := 1, BIT_ONS[1] := 1);
   SucroseCIP_RINGMAIN_REMOTE : CIP_REMOTE := (BIT_ONS[0] := 1, BIT_ONS[1] := 1);
   SucroseCIP_RUNNING : BOOL;
   SucroseCIP_SeatLift_Pulsing : BOOL;
   SucroseCIP_TK230101_REMOTE : CIP_REMOTE := (BIT_ONS[0] := 1, BIT_ONS[1] := 1);
   SucroseCIP_TK230201_REMOTE : CIP_REMOTE := (BIT_ONS[0] := 1, BIT_ONS[1] := 1);
   SucroseCIP_TK230301_REMOTE : CIP_REMOTE := (BIT_ONS[0] := 1, BIT_ONS[1] := 1);
   SucroseCIP_TT : BOOL;
   SucroseDischarge : Area_Program := (TMR_Alarm[0].PRE := 5000, TMR_Alarm[3].PRE := 30000, TMR_Logic[0].PRE := 28800000, TMR_Logic[1].PRE := 5000, TMR_Logic[2].PRE := 5000, TMR_Logic[3].PRE := 5000, TMR_Logic[4].PRE := 5000, TMR_Logic[6].PRE := 2000, TMR_Logic[7].PRE := 2000, TMR_Logic[8].PRE := 2000, TMR_Logic[9].PRE := 1000, TMR_Logic[10].PRE := 1000);
        .BIT_LOGIC[0].2   // PATH TO P_23_01_01 ENABLED
        .BIT_LOGIC[0].0   // SUCROSE HEADER ENABLED
        .BIT_LOGIC[0].3   // PATH TO P_23_01_02 ENABLED
        .BIT_LOGIC[0].1   // SUCROSE HEADER ACTIVE
        .BIT_LOGIC[0].5   // LATCH PATH TO P_23_01_02
        .BIT_LOGIC[0].4   // LATCH PATH TO P_23_01_01
        .BIT_LOGIC[0].7   // PATH TO P_23_01_02 OK
        .BIT_LOGIC[0].6   // PATH TO P_23_01_01 OK
        .BIT_LOGIC[0].12   // SUCROSE HEADER PURGE WATER ENABLED
        .TMR_LOGIC[5].DN   // SUCROSE HEADER PURGE WATER ENABLED
        .TMR_LOGIC[5]   // SUCROSE HEADER WATER PURGE TOTALIZER TIMER
        .BIT_HMI[0].4   // HMI SUCROSE HEADER PURGE WATER PUSHBUTTON
        .BIT_HMI[0].0   // HMI SUCROSE HEADER ENABLED PUSHBUTTON PRESSED
        .TMR_LOGIC[6]   // TK_23_01_01 PRIME UNLATCH TIMER
        .TMR_LOGIC[2].DN   // TK_23_03_01 PRIME ENABLED FOR P_23_01_01 PATH
        .TMR_LOGIC[7]   // TK_23_02_01 PRIME UNLATCH TIMER
        .TMR_LOGIC[8]   // TK_23_03_01 PRIME UNLATCH TIMER
        .BIT_LOGIC[0].8   // PRIME ENABLED ON AT LEAST ONE PATH
        .TMR_LOGIC[0]   // 8 HOUR TIMER FOR EACH DISCHARGE PATH
        .BIT_ALARM[0].0   // BOTH PATHS HAVE ALARMS ACTIVE ALARM LATCH
        .BIT_ALARM[0].1   // SUCROSE HEADER HIGH PRESSURE ALARM LATCH
        .BIT_ALARM[0].2   // SUCROSE HEADER LOW PRESSURE ALARM LATCH
        .BIT_ALARM[0].3   // SUCROSE HEADER LOW FLOW ALARM LATCH
        .TMR_ALARM[0]   // BOTH PATHS HAVE ALARMS ACTIVE TIMER
        .TMR_ALARM[1]   // SUCROSE HEADER HIGH PRESSURE ALARM TIMER
        .TMR_ALARM[2]   // SUCROSE HEADER LOW PRESSURE ALARM TIMER
        .TMR_ALARM[3]   // SUCROSE HEADER LOW FLOW ALARM TIMER
        .TMR_LOGIC[1]   // SUCROSE HEADER ACTIVE TIMER DELAY FOR PUMP START
        .TMR_LOGIC[2]   // TK_23_01_01 PRIME FROM TANK OUTLET TO DISCHARGE MANIFOLD
        .TMR_LOGIC[3]   // TK_23_02_01 PRIME FROM TANK OUTLET TO DISCHARGE MANIFOLD
        .TMR_LOGIC[4]   // TK_23_03_01 PRIME FROM TANK OUTLET TO DISCHARGE MANIFOLD
        .BIT_HMI[0].1   // HMI SUCROSE HEADER PATH SELECTION TO P_23_01_01 PUSHBUTTON PRESSED
        .BIT_HMI[0].2   // HMI SUCROSE HEADER PATH SELECTION TO P_23_01_02 PUSHBUTTON PRESSED
   SucroseFiltration : Area_Program := (BIT_Comment := 1, TMR_Alarm[0].PRE := 30000, TMR_Alarm[1].PRE := 30000, TMR_Alarm[2].PRE := 30000, TMR_Alarm[4].PRE := 30000, TMR_Alarm[5].PRE := 30000, TMR_Alarm[6].PRE := 30000, TMR_Alarm[7].PRE := 30000, TMR_Alarm[8].PRE := 30000, TMR_Alarm[9].PRE := 30000, TMR_Alarm[10].PRE := 30000, TMR_Alarm[11].PRE := 30000, TMR_Alarm[12].PRE := 30000, TMR_Alarm[13].PRE := 30000, TMR_Alarm[14].PRE := 30000, TMR_Alarm[15].PRE := 30000, CTR_Logic[0].DN := 1, CTR_Logic[1].DN := 1, CTR_Logic[2].DN := 1, CTR_Logic[3].DN := 1, CTR_Logic[4].DN := 1, CTR_Logic[5].DN := 1, CTR_Logic[6].DN := 1, CTR_Logic[7].DN := 1, STATUS_HMI[1] := 7, STATUS_HMI[2] := 7, STATUS_HMI[3] := 7, STATUS_HMI[4] := 7);
